// ---- POUs/FB/FB_Licznik.TcPOU
FUNCTION_BLOCK FB_Licznik 
VAR_INPUT
	c_inkrement : BOOL; // sygnal z czujnika
	czas : TIME; // określamy czas, który funkcja czeka po wykryciu butelki,... aby wyeliminowac drgania styków itd. 
END_VAR
VAR_OUTPUT
	c_stan: INT;
END_VAR
VAR
	timer1: TON;
	timer2: TON;
	zbocze	:R_TRIG;
	c_stanpomoc: INT;
END_VAR

c_stanpomoc:=c_stan;

//WHILE c_inkrement:= TRUE DO 					///to może być nie potrzbne 
	timer1(IN := c_inkrement, PT :=T#0.1S);
	zbocze(CLK := timer1.IN);
	IF zbocze.Q THEN
		c_stan:=c_stan+1;
	END_IF		
//END_WHILE

IF c_stan>c_stanpomoc THEN
	timer2(IN := TRUE, PT := czas);
	zbocze(CLK := timer2.IN);
END_IF
c_stanpomoc:=c_stan;

IF GVL_GLOBAL.reset_licznik:= TRUE THEN
	c_stan:=0;
END_IF

END_FUNCTION_BLOCK

// ---- POUs/RecipeManager/RecipeManagement.TcPOU
PROGRAM RecipeManagement
VAR
	fbRecipeManCommands 	: RecipeManCommands; (* Recipe Manager *)
	
	bInit 					: BOOL := TRUE;
	
	nLastError 				: DWORD; (* Error from Recipe Manager *)
	nRecipeCount 			: INT;
	
	sRecipeDef 				: STRING := 'Recipes'; (* current recipe definition *)
	sRecipe 				: STRING; (*Selected recipe *)
	nPreviousIndex			: INT; (* Previous selected index *)
	nPreviousSelectionIndex	: INT := -1; (* *)
	bReload 				: BOOL; (* Refresh recipes from files *)
	fbSaveVariablesTrigger	: R_TRIG;
	bSaveVariables			: BOOL;
	nSelectionIndexInList 	: INT;
	nCount					: INT;
	bReloadValues			: BOOL;
END_VAR

(* Initialization *)
IF bInit THEN
	(* Save the number of recipes in the specified recipe definition in a globar variable.*)
	GVL_RecipeTable.nRecipeCount := fbRecipeManCommands.GetRecipeCount(sRecipeDef);
	
	(* Empty all arrays *)
	FOR nCount := 0 TO cMaxTableRows DO
		GVL_RecipeTable.aRecipeNames[nCount] := '';
		GVL_RecipeTable.aVariableNames[nCount] := '';
		GVL_RecipeTable.aVariableValues[nCount] := '';
	END_FOR
	
	(* save all recipe names of the default recipe definition in an array *)
	fbRecipeManCommands.GetRecipeNames(	sRecipeDef,
										ADR(GVL_RecipeTable.aRecipeNames),
										10,
										GVL_RecipeTable.nRecipeIndex);
										
	GVL_RecipeTable.nRecipeSelectionIndex := -1;
	nPreviousSelectionIndex := -1;
	
	bInit := FALSE;
END_IF

(* Count all recipes in the defined recipe definition *)
nRecipeCount := fbRecipeManCommands.GetRecipeCount(sRecipeDef);
nLastError := fbRecipeManCommands.GetLastError();

(* Scroll position of the recipe list has changed. *)
IF GVL_RecipeTable.nRecipeIndex <> nPreviousIndex THEN
	fbRecipeManCommands.GetRecipeNames(	sRecipeDef,
										ADR(GVL_RecipeTable.aRecipeNames),
										10,
										GVL_RecipeTable.nRecipeIndex);
	nPreviousIndex := GVL_RecipeTable.nRecipeIndex;
END_IF

(* Selection of the current recipe has changed *)
IF GVL_RecipeTable.nRecipeSelectionIndex <> nPreviousSelectionIndex OR bReloadValues THEN
	nPreviousSelectionIndex := GVL_RecipeTable.nRecipeSelectionIndex;
	nSelectionIndexInList := GVL_RecipeTable.nRecipeSelectionIndex - GVL_RecipeTable.nRecipeIndex;
	
	(* Get the selected recipe name *)
	IF nSelectionIndexInList >= 0 AND nSelectionIndexInList < 10 THEN
		sRecipe := GVL_RecipeTable.aRecipeNames[nSelectionIndexInList];
	END_IF
	
	fbRecipeManCommands.GetRecipeValues(sRecipeDef,
										sRecipe,
										ADR(GVL_RecipeTable.aVariableValues),
										10,
										GVL_RecipeTable.nVariableIndex,
										80);
										
	fbRecipeManCommands.GetRecipeVariableNames(	sRecipeDef,
												sRecipe,
												ADR(GVL_RecipeTable.aVariableNames),
												10,
												GVL_RecipeTable.nVariableIndex);
	
	bReloadValues := FALSE;
END_IF

(* Reload the recipe list from the file system *)
IF bReload THEN
	
	fbRecipeManCommands.ReloadRecipes(sRecipeDef);
	bInit := TRUE;
	bReload := FALSE;
END_IF

(* Save the edited values into the recipe *)
fbSaveVariablesTrigger(CLK := bSaveVariables);
IF fbSaveVariablesTrigger.Q THEN
	fbRecipeManCommands.SetRecipeValues(sRecipeDef,
										sRecipe,
										ADR(GVL_RecipeTable.aVariableValues),
										10,
										GVL_RecipeTable.nVariableIndex);	
	bSaveVariables := FALSE;
END_IF

END_PROGRAM

// ---- POUs/Eventy/P_EventsSimple.TcPOU
//==================================================================================================
//							Beckhoff Automation Poland
//									5.2.2016
//		Program sluzy do przesylania globalnych tablic alarmow, ostrzezen i komunikatow do Event Loggera
//  v1.3	|| TC v 3.1.4020.28		|| - poprawki w MESSAGE, dodatkowe komentarze
//  v1.3	|| TC v 3.1.4020.28		|| - kosmetyka
//  v1.2	|| TC v 3.1.4020.28		|| - dodanie MESSAGE
//  v1.1 	|| TC v 3.1.4020.14 	|| - dodanie wersjonowania, komentarzy
// 	v1.0 	|| TC v 3.1.4020.0 		|| - pierwsza wersja
//==================================================================================================
PROGRAM P_EventsSimple
VAR
	fbAlarms				: FB_SimpleEventLog;								// Logowanie alarmow
	fbWarnings				: FB_SimpleEventLog;								// Logowanie ostrzezen
	fbMessage				: FB_SimpleEventLog;								// Logowanie komunikatow
	fbRead1					: FB_AdsReadEvents;									// Odczyt tablicy jezyk polski
	fbRead2					: FB_AdsReadEvents;									// Odczyt tablicy jezyk angielski
	fbRead3					: FB_AdsReadEvents;									// Odczyt tablicy jezyk niemiecki
	fbClear					: ADSCLEAREVENTS;									// Czyszczenie aktywnych alarmow
	MSG_ALARM_ListQuit		: ARRAY[FIRST_MESSAGE..LAST_MESSAGE] OF BOOL;		// Tablica nieuzywana - wymaga potwierdzenia przy usuwaniu
	MSG_MESSAGE_ListQuit	: ARRAY[FIRST_MESSAGE..LAST_MESSAGE] OF BOOL;		// Tablica nieuzywana - wymaga potwierdzenia przy usuwaniu
	MSG_WARNING_ListQuit	: ARRAY[FIRST_MESSAGE..LAST_MESSAGE] OF BOOL;		// Tablica nieuzywana - wymaga potwierdzenia przy usuwaniu
END_VAR

(*
	TCEVENTCLASS_NONE			:=0,	No class
	TCEVENTCLASS_MAINTENANCE	:=1,	Maintenance hint
	TCEVENTCLASS_MESSAGE		:=2,	Message
	TCEVENTCLASS_HINT			:=3,	Hint
	TCEVENTCLASS_STATEINFO		:=4,	State information
	TCEVENTCLASS_INSTRUCTION	:=5,	Instruction
	TCEVENTCLASS_WARNING		:=6,	Warning
	TCEVENTCLASS_ALARM			:=7,	Alarm
	TCEVENTCLASS_PARAMERROR		:=8	 	Parameter error
*)
fbClear(	bClear			:= TRUE,
			iMode			:= TCEVENTLOGIOFFS_CLEARALL);

fbAlarms(	Init			:= TRUE,
			SourceId		:= 1,
			Class			:= TCEVENTCLASS_ALARM,
			QuitRequired	:= FALSE,
			adrAlarmArray	:= ADR(MSG_ALARM_List),
			adrQuitArray	:= ADR(MSG_ALARM_ListQuit));
	
fbWarnings(	Init			:= TRUE,
			SourceId		:= 2,
			Class			:= TCEVENTCLASS_WARNING,
			QuitRequired	:= FALSE,
			adrAlarmArray	:= ADR(MSG_WARNING_List),
			adrQuitArray	:= ADR(MSG_WARNING_ListQuit));

fbMessage(	Init			:= TRUE,
			SourceId		:= 3,
			Class			:= TCEVENTCLASS_MESSAGE,
			QuitRequired	:= FALSE,
			adrAlarmArray	:= ADR(MSG_MESSAGE_List),
			adrQuitArray	:= ADR(MSG_MESSAGE_ListQuit));
			
// Odczyt w kilku jezykach
fbRead1(	bReadEvents		:= TRUE,
			nLanguageId		:= 1045,
			tRefreshTime	:= T#1S);

fbRead2(	bReadEvents		:= TRUE,
			nLanguageId		:= 1033,
			tRefreshTime	:= T#1S);

fbRead3(	bReadEvents		:= TRUE, 
			nLanguageId		:= 1031, 
			tRefreshTime	:= T#1S);
			
// Wybor aktualnego jezyka wyswietlania - przepisanie do tablicy odpowiedniej tablicy
// Uwaga j. polski bez polskich znakow
IF VisuElemsWinControls.CURRENTLANGUAGE		= 'en' THEN
	aEventsSimple			:= fbRead2.aEvents;
ELSIF VisuElemsWinControls.CURRENTLANGUAGE	= 'de' THEN
	aEventsSimple			:= fbRead3.aEvents;
ELSE
	aEventsSimple			:= fbRead1.aEvents;	
END_IF;

END_PROGRAM

// ---- POUs/Eventy/FB_SimpleEventLog.TcPOU
//==================================================================================================
//							Beckhoff Automation Poland
//									22.12.2016
//	Program glowny dla zdarzen wersji advanced
// 	v1.1	|| TC v 3.1.4020.28		|| - idx, ARRAY_LBOUND, ARRAY_UBOUND --> Zmiana typu z UDINT na DINT
// 	v1.0	|| TC v 3.1.4020.28		|| - pierwsza wersja - 13.10.2004, Author:			Dirk Nordberg (BECKHOFF INDUSTRIE ELEKTRONIK)
// Description: Function block to control the EventLogger
// 	Messages can be activated or deactivated through an array of bool.
// 	The subscription of the array is equivalent to EventID from EventLogger.
// 	Funtion block will be initialized with Init flag, then the busy flag is set true. 
// 
// 	Revision:	1.4
// 	History:		13.10.2004	Ng	start coding
// 					17.04.2005	MK	runtime optimized
// 					07.07.2005	MK	short puls BF
// 				    29.11.2010 	MiB  quittierungspflichtige Merker funktionieren nun wieder
///                 21.06.2013  TV   change : data type for pointer address from uint to pointer of int 
//==================================================================================================
///****************************************************************************************
///Name:				FB_SimpleEventLog
///Date:				13.10.2004
// 

FUNCTION_BLOCK FB_SimpleEventLog
VAR_INPUT
	/// Rising flag starts the initialization 
	Init: BOOL;
	/// Number of the source Id 
	SourceId: UINT;
	/// Alarm error class 
	Class: UINT;
	/// Activate or deaktivate confirmation 
	QuitRequired: BOOL;
	/// Adress of the array for the messages 
	adrAlarmArray: POINTER TO BOOL;
	/// ...with constant boundaries ARRAY_LBOUND to ARRAY_UBOUND for array size 
	adrQuitArray: POINTER TO BOOL;
END_VAR
VAR_OUTPUT
	Busy: BOOL;
	Err: BOOL;
	ErrId: UDINT;
END_VAR
VAR CONSTANT
	ARRAY_LBOUND: DINT := FIRST_MESSAGE;
	ARRAY_UBOUND: DINT := LAST_MESSAGE;
	TCEVENTDATAFORMATSTRING: STRING := ' ';
	STATE_INIT: INT := 0;
	STATE_IDLE: INT := 1;
	STATE_RESET_EVENT: INT := 2;
	STATE_QUIT_EVENT: INT := 3;
	STATE_RESET_END: INT := 4;
	STATE_WAIT: INT := 5;
END_VAR
VAR
	state: INT;
	///{flag nowatch on }
	bReady: BOOL := TRUE;
	nMsgHasChanged: DINT;
	bEvtState: ARRAY[ARRAY_LBOUND..ARRAY_UBOUND] OF BOOL;
	event: ARRAY[ARRAY_LBOUND..ARRAY_UBOUND] OF ADSLOGEVENT;
	idx: DINT;
	CfgEvent: TcEvent;
	bWait: BOOL;
	ptAlarm: POINTER TO BOOL;
	ptQuit: POINTER TO BOOL;
	RT_Init: R_TRIG;
END_VAR

nMsgHasChanged := MEMCMP(ADR(bEvtState), adrAlarmArray, SIZEOF(bEvtState));

RT_Init(CLK:=Init);

CASE State OF
	STATE_INIT:		(* Set the parameter for TcEvent *)
		Err := FALSE;
		ErrId :=0;
		Busy := FALSE;
		CfgEvent.Prio := 0;
		CfgEvent.DataFormatStrAddress := ADR(TCEVENTDATAFORMATSTRING);
		// CfgEvent.Flags := TCEVENTFLAG_LOG OR TCEVENTFLAG_SRCID OR TCEVENTFLAG_PRIOCLASS OR TCEVENTFLAG_FMTSELF OR 16#1000;
		// MiB 2015.10.07 Flags changed -> now the class is defined here and not in Event config file.
		CfgEvent.Flags := TCEVENTFLAG_LOG OR TCEVENTFLAG_SRCID;
		CfgEvent.StreamType := TCEVENTSTREAM_SIMPLE;
		CfgEvent.ProgId := 'TcEventFormatter.TcXmlFormatter';
		CfgEvent.SourceId := SourceId;
			CfgEvent.Class := Class ;
		CfgEvent.bQuitRequired := QuitRequired;
		FOR idx := ARRAY_LBOUND TO ARRAY_UBOUND BY 1 DO
			CfgEvent.Id := DINT_TO_UDINT(idx);
			event[idx](NETID:='', PORT:=110, Event:=FALSE , EventQuit:=FALSE,
				 EventConfigData:=CfgEvent, FbCleanup:=FALSE, TMOUT:=t#1s);
		END_FOR;
		State := STATE_IDLE;

	STATE_IDLE:
		(* nothing to do *)
		IF nMsgHasChanged = 0
			AND  NOT QuitRequired
			AND bReady = TRUE
			AND NOT RT_Init.Q THEN
			RETURN;
		END_IF

		IF adrAlarmArray <> 0 THEN
			ptAlarm := adrAlarmArray;
			IF CfgEvent.bQuitRequired AND adrQuitArray <> 0 THEN
				ptQuit := adrQuitArray;
				FOR idx := ARRAY_LBOUND TO ARRAY_UBOUND BY 1 DO
					event[idx](Event:=ptAlarm^, EventQuit:=ptQuit^);
					ptAlarm := ptAlarm + 1;
					ptQuit := ptQuit + 1;
				END_FOR;
				bReady := TRUE;
			ELSE
				bReady := TRUE;
				FOR idx := ARRAY_LBOUND TO ARRAY_UBOUND BY 1 DO
					event[idx](Event:=ptAlarm^);
					IF (NOT (ptAlarm^ = TRUE
							AND event[idx].Event = TRUE		(* event is set/on *)
							AND event[idx].Quit = FALSE
							AND event[idx].EventState = TCEVENTSTATE_SIGNALED)
						AND NOT (ptAlarm^ = FALSE
							AND event[idx].Event = FALSE		(* event is reset/off *)
							AND event[idx].Quit = TRUE
							AND event[idx].EventState = TCEVENTSTATE_INVALID)) THEN
						bReady := FALSE;
					END_IF
					ptAlarm := ptAlarm + 1;
				END_FOR;

				(* copy the status *)
				IF bReady THEN
					MEMCPY(ADR(bEvtState), adrAlarmArray, SIZEOF(bEvtState));
				END_IF

			END_IF
		END_IF

		IF RT_Init.Q THEN
			Busy := TRUE;
			State := STATE_RESET_EVENT;
		END_IF

	STATE_RESET_EVENT:(*---------------------------------- clear messages ----------------------------------------*)
		FOR idx := ARRAY_LBOUND TO ARRAY_UBOUND BY 1 DO
			IF event[idx].EventState = TCEVENTSTATE_SIGNALED THEN
				event[idx](Event:=FALSE, EventQuit:= FALSE, FbCleanup:= FALSE, TMOUT:= t#1s);
				IF event[idx].Err THEN
					Err := TRUE;
					ErrId := event[idx].ErrId;
					IF event[idx].ErrId = 1282 THEN	(* Message Router: mailbox full *)
						event[idx](Event:=FALSE, EventQuit:= FALSE, FbCleanup:= FALSE);
						RETURN;
					END_IF
				END_IF
			END_IF;
		END_FOR;
		State := STATE_QUIT_EVENT;

	STATE_QUIT_EVENT:(*---------------------------------- quit messages ----------------------------------------*)
		FOR idx := ARRAY_LBOUND TO ARRAY_UBOUND BY 1 DO
			IF event[idx].EventState = TCEVENTSTATE_SIGNALED THEN
				event[idx](Event:=FALSE, EventQuit:= TRUE, FbCleanup:= FALSE, TMOUT:= t#1s);
				IF event[idx].Err THEN
					Err := TRUE;
					ErrId := event[idx].ErrId;
					IF event[idx].ErrId = 1282 THEN	(* Message Router: mailbox full *)
						event[idx](Event:=FALSE, EventQuit:= FALSE, FbCleanup:= FALSE);
						RETURN;
					END_IF
				END_IF
			END_IF;
		END_FOR;
		State := STATE_RESET_END;

	STATE_RESET_END:
		bWait := FALSE;
		FOR idx := ARRAY_LBOUND TO ARRAY_UBOUND BY 1 DO
			event[idx](Event:=FALSE, EventQuit:= FALSE, FbCleanup:= FALSE);
			IF event[idx].EventState = TCEVENTSTATE_SIGNALED THEN
				bWait := TRUE;
			END_IF
		END_FOR;
		IF NOT bWait THEN
			State := STATE_INIT;
		END_IF

END_CASE

END_FUNCTION_BLOCK

// ---- POUs/FB/FB_INV000_MX2_Alarm.TcPOU
FUNCTION_BLOCK FB_INV000_MX2_Alarm
VAR_INPUT
	Enable							:BOOL;	
	Fault_Monitor_1_Inverter_Status	:UINT;
	Fault_Monitor_1_Cause			:UINT;	
	Status							:WORD;	

END_VAR
VAR_OUTPUT
	ENO								:BOOL;	
	Alarm_Status					:STRING[256];
	Alarm_Fault						:STRING[256];	

END_VAR
VAR
	tmp_Status						:uWORD_BOOL_MX2;
END_VAR

///FB ON///
ENO:=Enable;

///Status extraction///
	tmp_Status.ch := Status;

//If MX2 has an fault the latest fault will be outputted//
IF tmp_Status.bits[3]=TRUE THEN
	
//MX2 Inverter fault factor list name//
CASE Fault_Monitor_1_Cause OF
	00 : 
		Alarm_Fault:='No trip factor';	
	01 : 
		Alarm_Fault:='Overcurrent protection during constant speed';
   	02 : 
		Alarm_Fault:='Overcurrent protection during deceleration';
	03 : 
		Alarm_Fault:='Overcurrent protection during acceleration';
	04 : 
		Alarm_Fault:='Overcurrent protection during stop';
	05 : 
		Alarm_Fault:='Overload protection';
	06 : 
		Alarm_Fault:='Braking resistor overload protection';
	07 : 
		Alarm_Fault:='Overvoltage protection';
	08 : 
		Alarm_Fault:='EEPROM error';
	09 : 
		Alarm_Fault:='Undervoltage protection';
	10 : 
		Alarm_Fault:='Current detector error';
	11 : 
		Alarm_Fault:='CPU error';
	12 : 
		Alarm_Fault:='External trip';
	13 : 
		Alarm_Fault:='USP error';
	14 : 
		Alarm_Fault:='Grounding protection';
	15 : 
		Alarm_Fault:='Incoming overvoltage protection';
	21 : 
		Alarm_Fault:='Abnormal temperature';
	25 : 
		Alarm_Fault:='Main circuit error';
	30 : 
		Alarm_Fault:='Driver error';
	35 : 
		Alarm_Fault:='Thermistor error';
	36 : 
		Alarm_Fault:='Brake error';
	37 : 
		Alarm_Fault:='Emergency shutoff';
	38 : 
		Alarm_Fault:='Overload protection in a low speed range';
	40 : 
		Alarm_Fault:='Digital operator connection error';
	41 : 
		Alarm_Fault:='Modbus communication (Modbus-RTU) error';
	43..45 : 
		Alarm_Fault:='Internal data error';
	50..69 : 
		Alarm_Fault:='Internal data error';	
	80 : 
		Alarm_Fault:='Encoder disconnection';
	81 : 
		Alarm_Fault:='Overspeed';
	83 : 
		Alarm_Fault:='Position control range trip';
	

		
END_CASE;

//MX2 Inverter status at fault occur//


	CASE Fault_Monitor_1_Inverter_Status OF
    	0 : 
			Alarm_Status:='During reset';
		1 : 
			Alarm_Status:='During stop';
		2 : 
			Alarm_Status:='During deceleration';
		3 : 
			Alarm_Status:='At a constant speed';
		4 : 
			Alarm_Status:='During acceleration';
		5 : 
			Alarm_Status:='Operates at frequency = 0';
		6 : 
			Alarm_Status:='During startup';
		7 : 
			Alarm_Status:='DB active (DC injection braking active)';
		8 : 
			Alarm_Status:='During overload limit';
		
	END_CASE;
ELSE
	Alarm_Fault:='No trip factor';	
	Alarm_Status:='--';
	
END_IF;

END_FUNCTION_BLOCK

// ---- POUs/FB/FB_INV003_MX2_ECT.TcPOU
FUNCTION_BLOCK FB_INV003_MX2_ECT
VAR_INPUT
	Output_Frequency_Monitor						:UINT;
	Enable											:BOOL;
	Fwd												:BOOL;	
	Rev												:BOOL;	
	Fault_Reset										:BOOL;	
	Frequency_in									:REAL;	
	Acceleration									:REAL;		
	Deceleration									:REAL;	
END_VAR
VAR_OUTPUT
	ENO												:BOOL;
	Frequency_out									:REAL;	
	During_Fwd										:BOOL;
	During_Rev										:BOOL;	
	Fault											:BOOL;		
	Warning											:BOOL;		
	Remote											:BOOL;	
	Freq_Match										:BOOL;	
	Connection_Error								:BOOL;		
END_VAR
VAR
	tmp_freq_in_real								:REAL;
	tmp_freq_in_int									:UINT;			
	tmp_freq_out_real								:REAL;			
	tmp_freq_out_int								:UINT;			
	tmp_acc_real									:REAL;				
	tmp_acc_int										:INT;				
	tmp_dec_real									:REAL;				
	tmp_dec_int										:INT;		
	tmp_Command										:uWORD_BOOL_MX2;			
	tmp_Status										:uWORD_BOOL_MX2;	
END_VAR
VAR_IN_OUT
	Command												:WORD;	
	Frequency_Reference									:UINT;	
	F002_1st_Acceleration								:UDINT;		
	F003_1st_Deceleration								:UDINT;		
	Status												:WORD;	
END_VAR

///Status extraction///
	tmp_Status.ch := Status;
	During_Fwd := tmp_Status.bits[0];
	During_Rev := tmp_Status.bits[1];
	Fault := tmp_Status.bits[3];
	Warning := tmp_Status.bits[7];
	Remote := tmp_Status.bits[9];
	Freq_Match := tmp_Status.bits[12];
	Connection_Error := tmp_Status.bits[15];

///Command extraction///
IF Enable THEN;
	tmp_Command.bits[0] := Fwd;
	tmp_Command.bits[1] := Rev;
	ENO:=TRUE;
ELSE
	tmp_Command.bits[0] := FALSE;
	tmp_Command.bits[1] := FALSE;
	ENO:=FALSE;
END_IF;
	tmp_Command.bits[7] := Fault_Reset;
	Command := tmp_Command.ch;

///Frequence form a REAL value///
IF Frequency_in>0.01 THEN;
	tmp_freq_in_real:=Frequency_in*100;
	tmp_freq_in_int:=REAL_TO_UINT(tmp_freq_in_real);
	Frequency_Reference:=tmp_freq_in_int;
END_IF;

//Convert Output_Frequency_Monitor to a REAL value//
	tmp_freq_out_int:=Output_Frequency_Monitor;
	tmp_freq_out_real:=UINT_TO_REAL(tmp_freq_out_int);
	Frequency_out:=tmp_freq_out_real/100.0;
	
//Acceleration/Deceleration Time  in REAL value//
IF Acceleration>0.01 THEN;
	tmp_acc_real:=Acceleration*100;
	tmp_acc_int:=REAL_TO_INT(tmp_acc_real);
	F002_1st_Acceleration:=tmp_acc_int;
END_IF;

IF Deceleration>0.01 THEN;
	tmp_dec_real:=Deceleration*100;
	tmp_dec_int:=REAL_TO_INT(tmp_dec_real);
	F003_1st_Deceleration:=tmp_dec_int;
END_IF;

END_FUNCTION_BLOCK

// ---- POUs/Programy/Hbot/AxisOnline/POUsAxisOnline/AX5000/FB_AxisDiag_1.TcPOU
//==================================================================================================
//							Beckhoff Automation Poland
//								23.05.2018
//					Blok do diagnostyki osi
// 	v1.1	|| TC v 3.1.4022.16	|| - optymalizacja kodu
// 	v1.0	|| TC v 3.1.4020.0	|| - pierwsza wersja
//==================================================================================================
FUNCTION_BLOCK FB_AxisDiag_1
VAR_INPUT
	IPCNetID							: T_AmsNetId; 	(* AmsNetId of the IPC *)
	Timeout								: TIME := DEFAULT_ADS_TIMEOUT;
	Reset								: BOOL;
	GetDiag								: BOOL;
END_VAR
VAR_IN_OUT
	Axis	 							: AXIS_REF;
	stAX5000Diag						: ST_AX5000Diag;
END_VAR
VAR_OUTPUT
	Error								: BOOL;
	AdsErrId							: UINT;
	SercosErrId							: UINT;
	ResetAct							: BOOL;
	DiagAct								: BOOL;
	Busy								: BOOL;
END_VAR
VAR
	iState								: INT;
	iSubState							: INT;
	GetDriveRef							: BOOL;
	DriveRef								: ST_DriveRef; (* contains sNetID of EcMaster, nSlaveAddr of EcDrive, nDriveNo of EcDrive, either preset or read from NC *)
	AxisID								: UDINT;

	C1DErrorPrev							: BOOL;
	WcStateErrorPrev						: BOOL;
	AxisErrorPrev							: BOOL;
	OperationalPrev						: BOOL;
	ResetPrev							: BOOL;
	GetDiagPrev							: BOOL;

	fbSoERead							: FB_SoERead;
	fbDiagMessage 						: FB_SoEReadDiagMessage;
	fbClassXDiag							: FB_SoEReadClassXDiag;
	fbDiagNumber						: FB_SoEReadDiagNumber;
	fbDiagNumberList						: FB_SoEReadDiagNumberList;

	fbReset								: FB_SoEReset;
	fbDelay								: TON;
	fbGetSlaveState 						: FB_EcGetSlaveState;
	fbReqSlaveState 						: FB_EcReqSlaveState;
	fbNcReset 							: MC_Reset;

	fbAdsRead							: ADSREAD;
	readBuffer							: ARRAY[0..9] OF BYTE;
	Ids									: T_AmsNetIdArr;
	strSoEString							: ST_SoE_String;
END_VAR
VAR CONSTANT
	NCIDXG_AXPARMS					: UDINT := 16#00004000;	(* Axis with ID: Parameter 			*)
	NCIDXO_AXP_HWAMSADDR			: UDINT := 16#00000031;
END_VAR

stAX5000Diag.bOperational	:= Axis.NcToPlc.StateDWord.0;
stAX5000Diag.bC1DError	 	:= Axis.NcToPlc.StateDWord.28;
stAX5000Diag.bWcStateError 	:= Axis.NcToPlc.StateDWord.30;
stAX5000Diag.bAxisError		:= Axis.NcToPlc.StateDWord.31;
stAX5000Diag.iAxisErrorCode	:= Axis.NcToPlc.ErrorCode;

CASE iState OF
0:	(* idle *)
	GetDriveRef 	:= (DriveRef.nSlaveAddr = 0);

	IF GetDriveRef THEN
		Busy			:= TRUE;
		Error			:= FALSE;
		AdsErrId		:= 0;
		SercosErrId		:= 0;
		iState 			:= 1;
		iSubState		:= 0;
		AxisID 			:= Axis.NcToPlc.AxisId;

	ELSIF Reset AND NOT ResetPrev THEN
		Busy			:= TRUE;
		ResetAct		:= TRUE;
		ResetPrev		:= Reset;
		Error			:= FALSE;
		AdsErrId		:= 0;
		SercosErrId		:= 0;
		iState 			:= 2;
		iSubState		:= 0;
		AxisID 			:= Axis.NcToPlc.AxisId;

	ELSIF GetDiag AND NOT GetDiagPrev OR
		(stAX5000Diag.bC1DError AND NOT C1DErrorPrev) OR (NOT stAX5000Diag.bC1DError AND C1DErrorPrev) (* rising/falling C1D *) OR
		(stAX5000Diag.bWcStateError AND NOT WcStateErrorPrev) OR (NOT stAX5000Diag.bWcStateError AND WcStateErrorPrev) (* rising/falling WcState *) OR
		(stAX5000Diag.bAxisError AND NOT AxisErrorPrev) OR (NOT stAX5000Diag.bAxisError AND AxisErrorPrev) (* rising/falling NcError *) OR
		(stAX5000Diag.bOperational AND NOT OperationalPrev) OR (NOT stAX5000Diag.bOperational AND OperationalPrev) (* rising/falling Enable *) THEN

		Busy			:= TRUE;
		DiagAct			:= TRUE;
		GetDiagPrev		:= GetDiag;
		Error			:= FALSE;
		AdsErrId		:= 0;
		SercosErrId		:= 0;
		iState 			:= 3;
		iSubState		:= 0;
		AxisID 			:= Axis.NcToPlc.AxisId;

		(* set/clear flags *)
		C1DErrorPrev		:= stAX5000Diag.bC1DError;
		WcStateErrorPrev	:= stAX5000Diag.bWcStateError;
		AxisErrorPrev		:= stAX5000Diag.bAxisError;
		OperationalPrev		:= stAX5000Diag.bOperational;

	ELSE
		ResetAct	:= FALSE;
		DiagAct		:= FALSE;
	END_IF

1:	(* get drive reference *)
	M_GetDriveRef();

2:	(* reset and state change *)
	M_Reset();

3:	(* get diag data *)
	M_GetDiagnosis();

END_CASE

(* clear latch *)
ResetPrev	:= ResetPrev AND Reset;
GetDiagPrev	:= GetDiagPrev AND GetDiag;

ACTION M_GetDiagnosis:
CASE iSubState OF
0:	fbClassXDiag(
		NetId		:= IPCNetID,
		Execute		:= TRUE,
		DiagClass 	:= 1,
		Timeout		:= DEFAULT_ADS_TIMEOUT,
		Axis		:= Axis,
	);

	IF NOT fbClassXDiag.Busy THEN
		fbClassXDiag(Execute:= FALSE,Axis := Axis);

		IF NOT fbClassXDiag.Error THEN
			stAX5000Diag.wClass1Diag	:= fbClassXDiag.ClassXDiag;
			stAX5000Diag.stClass1Diag	:= F_ConvWordToSTAX5000C1D(stAX5000Diag.wClass1Diag);
		ELSE
			Error			:= TRUE;
			AdsErrId		:= fbClassXDiag.AdsErrId;
			SercosErrId	:= fbClassXDiag.SercosErrId;
		END_IF
		iSubState	:= iSubState + 1;
	END_IF

1:	fbDiagMessage(
		NetId	:= IPCNetID,
		Execute	:= TRUE,
		Timeout	:= DEFAULT_ADS_TIMEOUT,
		Axis	:= Axis,
	);

	IF NOT fbDiagMessage.Busy THEN
		fbDiagMessage(Execute:= FALSE,Axis := Axis);

		IF NOT fbDiagMessage.Error THEN
			stAX5000Diag.strDiagMessage := LEFT(fbDiagMessage.DiagMessage.strData, UINT_TO_INT(fbDiagMessage.DiagMessage.iActualSize));
		ELSE
			Error			:= TRUE;
			AdsErrId		:= fbDiagMessage.AdsErrId;
			SercosErrId	:= fbDiagMessage.SercosErrId;
		END_IF
		iSubState	:= iSubState + 1;
	END_IF

2:	fbDiagNumber(
		NetId	:= IPCNetID,
		Execute	:= TRUE,
		Timeout	:= DEFAULT_ADS_TIMEOUT,
		Axis	:= Axis,
	);

	IF NOT fbDiagNumber.Busy THEN
		fbDiagNumber(Execute:= FALSE,Axis := Axis);

		IF NOT fbDiagNumber.Error THEN
			stAX5000Diag.iDiagNumber := fbDiagNumber.DiagNumber;
		ELSE
			Error			:= TRUE;
			AdsErrId		:= fbDiagNumber.AdsErrId;
			SercosErrId	:= fbDiagNumber.SercosErrId;
		END_IF
		iSubState	:= iSubState + 1;
	END_IF

3:	fbSoERead(
		NetId	:= IPCNetID,
		Execute	:= TRUE,
		Idn		:= 135,
		Element	:=16#44,
		pDstBuf	:=ADR(stAX5000Diag.wDriveStatus),
		BufLen	:=SIZEOF(stAX5000Diag.wDriveStatus),
		Timeout	:= DEFAULT_ADS_TIMEOUT,
		Axis	:= Axis,
	);

	IF NOT fbSoERead.Busy THEN
		fbSoERead(Execute:= FALSE,Axis := Axis);
		IF NOT fbSoERead.Error THEN
			stAX5000Diag.stDriveStatus := F_ConvWordToSTAX5000DriveStatus(stAX5000Diag.wDriveStatus);
			iSubState		:= iSubState + 1;
		ELSE
			Error			:= TRUE;
			AdsErrId		:= fbSoERead.AdsErrId;
			SercosErrId	:= fbSoERead.SercosErrId;
			iSubState		:= iSubState + 2;
		END_IF
	END_IF

4:	fbSoERead(
		NetId	:= IPCNetID,
		Execute	:= TRUE,
		Idn		:= stAX5000Diag.stDriveStatus.iActOpModeParNum,
		Element	:=16#44,
		pDstBuf	:=ADR(stAX5000Diag.stDriveStatus.eActOpMode),
		BufLen	:=SIZEOF(stAX5000Diag.stDriveStatus.eActOpMode),
		Timeout	:= DEFAULT_ADS_TIMEOUT,
		Axis	:= Axis,
	);

	IF NOT fbSoERead.Busy THEN
		fbSoERead(Execute:= FALSE,Axis := Axis);
		IF NOT fbSoERead.Error THEN
			;
		ELSE
			Error			:= TRUE;
			AdsErrId		:= fbSoERead.AdsErrId;
			SercosErrId	:= fbSoERead.SercosErrId;
		END_IF
		iSubState	:= iSubState + 1;
	END_IF

5:	fbGetSlaveState(
		sNetId		:= DriveRef.sNetId,
		nSlaveAddr	:= DriveRef.nSlaveAddr,
		bExecute	:= TRUE,
		tTimeout	:= DEFAULT_ADS_TIMEOUT,
	);

	IF NOT fbGetSlaveState.bBusy THEN
		fbGetSlaveState(bExecute:= FALSE);
		IF NOT fbGetSlaveState.bError THEN
			stAX5000Diag.stEcSlaveState := fbGetSlaveState.state;
			stAX5000Diag.stEcSlaveStateBits := F_ConvSlaveStateToBits(fbGetSlaveState.state);
		ELSE
			Error			:= TRUE;
			AdsErrId		:= UDINT_TO_UINT(fbGetSlaveState.nErrId);
		END_IF

		IF stAX5000Diag.stEcSlaveStateBits.bError THEN
			IF stAX5000Diag.stEcSlaveStateBits.bPreop THEN
				(* read S21 - IDN List of Invalid operation data for CP2 (Preop->SaveOp) *)
				MEMSET(ADR(stAX5000Diag.stCPxInvParamList), 0, SIZEOF(stAX5000Diag.stCPxInvParamList));
				stAX5000Diag.bPreopToSafeOpError := TRUE;
				stAX5000Diag.bSafeOpToOpError := FALSE;
				iSubState	:= iSubState + 1;
			ELSIF stAX5000Diag.stEcSlaveStateBits.bSafeOp THEN
				(* read S22 - IDN List of Invalid operation data for CP3 (SaveOp->Op) *)
				MEMSET(ADR(stAX5000Diag.stCPxInvParamList), 0, SIZEOF(stAX5000Diag.stCPxInvParamList));
				stAX5000Diag.bPreopToSafeOpError := FALSE;
				stAX5000Diag.bSafeOpToOpError := TRUE;
				iSubState	:= iSubState + 2;
			ELSE
				(* Skip S21 + S22 *)
				MEMSET(ADR(stAX5000Diag.stCPxInvParamList), 0, SIZEOF(stAX5000Diag.stCPxInvParamList));
				stAX5000Diag.bPreopToSafeOpError := FALSE;
				stAX5000Diag.bSafeOpToOpError := FALSE;
				iSubState	:= iSubState + 3;
			END_IF
		ELSE
			(* Skip S21 + S22 *)
			MEMSET(ADR(stAX5000Diag.stCPxInvParamList), 0, SIZEOF(stAX5000Diag.stCPxInvParamList));
			stAX5000Diag.bPreopToSafeOpError := FALSE;
			stAX5000Diag.bSafeOpToOpError := FALSE;
			iSubState	:= iSubState + 3;
		END_IF
	END_IF

6:	(* read S21 - IDN List of Invalid operation data for CP2 (Preop->SaveOp) *)
	fbSoERead(
		NetId	:= IPCNetID,
		Execute	:= TRUE,
		Idn		:= 21,
		Element	:=16#40,
		pDstBuf	:=ADR(stAX5000Diag.stCPxInvParamList),
		BufLen	:=SIZEOF(stAX5000Diag.stCPxInvParamList),
		Timeout	:= DEFAULT_ADS_TIMEOUT,
		Axis	:= Axis,
	);

	IF NOT fbSoERead.Busy THEN
		fbSoERead(Execute:= FALSE,Axis := Axis);
		IF NOT fbSoERead.Error THEN
			;
		ELSE
			Error			:= TRUE;
			AdsErrId		:= fbSoERead.AdsErrId;
			SercosErrId	:= fbSoERead.SercosErrId;
		END_IF
		iSubState	:= iSubState + 2;
	END_IF

7:	(* read S22 - IDN List of Invalid operation data for CP3 (SaveOp->Op) *)
	fbSoERead(
		NetId	:= IPCNetID,
		Execute	:= TRUE,
		Idn		:= 22,
		Element	:=16#40,
		pDstBuf	:=ADR(stAX5000Diag.stCPxInvParamList),
		BufLen	:=SIZEOF(stAX5000Diag.stCPxInvParamList),
		Timeout	:= DEFAULT_ADS_TIMEOUT,
		Axis	:= Axis,
	);

	IF NOT fbSoERead.Busy THEN
		fbSoERead(Execute:= FALSE,Axis := Axis);
		IF NOT fbSoERead.Error THEN
			;
		ELSE
			Error			:= TRUE;
			AdsErrId		:= fbSoERead.AdsErrId;
			SercosErrId	:= fbSoERead.SercosErrId;
		END_IF
		iSubState	:= iSubState + 1;
	END_IF

8:	fbDiagNumberList(
		NetId			:= IPCNetID,
		Execute			:= TRUE,
		Timeout			:= DEFAULT_ADS_TIMEOUT,
		pDiagNumber		:= ADR(stAX5000Diag.stDiagNumberList),
		Size			:= SIZEOF(stAX5000Diag.stDiagNumberList),
		Axis			:= Axis,
	);

	IF NOT fbDiagNumberList.Busy THEN
		fbDiagNumberList(Execute:= FALSE,Axis := Axis);

		IF fbDiagNumberList.Error THEN
			Error			:= TRUE;
			AdsErrId		:= fbDiagNumberList.AdsErrId;
			SercosErrId	:= fbDiagNumberList.SercosErrId;
		END_IF

		IF (stAX5000Diag.strMotorType = '') OR (stAX5000Diag.strDriveType = '') THEN
			iSubState	:= iSubState + 1;
		ELSE
			DiagAct	:= FALSE;
			iSubState	:= 0;
			iState		:= 0;
			Busy		:= FALSE;
		END_IF
	END_IF

9:	fbSoERead(
		NetId	:= IPCNetID,
		Execute	:= TRUE,
		Idn		:= P_0_IDN + 53,
		Element	:=16#44,
		pDstBuf	:=ADR(strSoEString),
		BufLen	:=SIZEOF(strSoEString),
		Timeout	:= DEFAULT_ADS_TIMEOUT,
		Axis	:= Axis,
	);

	IF NOT fbSoERead.Busy THEN
		fbSoERead(Execute:= FALSE,Axis := Axis);
		IF NOT fbSoERead.Error THEN
			MEMSET(ADR(stAX5000Diag.strMotorType),0,SIZEOF(stAX5000Diag.strMotorType));
			MEMCPY(ADR(stAX5000Diag.strMotorType),ADR(strSoEString.strData),MIN(SIZEOF(stAX5000Diag.strMotorType),strSoEString.iActualSize));
		ELSE
			Error			:= TRUE;
			AdsErrId		:= fbSoERead.AdsErrId;
			SercosErrId	:= fbSoERead.SercosErrId;
		END_IF
		iSubState	:= iSubState + 1;
	END_IF

10:	fbSoERead(
		NetId	:= IPCNetID,
		Execute	:= TRUE,
		Idn		:= P_0_IDN + 324,
		Element	:=16#44,
		pDstBuf	:=ADR(strSoEString),
		BufLen	:=SIZEOF(strSoEString),
		Timeout	:= DEFAULT_ADS_TIMEOUT,
		Axis	:= Axis,
	);

	IF NOT fbSoERead.Busy THEN
		fbSoERead(Execute:= FALSE,Axis := Axis);
		IF NOT fbSoERead.Error THEN
			MEMSET(ADR(stAX5000Diag.strDriveType),0,SIZEOF(stAX5000Diag.strDriveType));
			MEMCPY(ADR(stAX5000Diag.strDriveType),ADR(strSoEString.strData),MIN(SIZEOF(stAX5000Diag.strDriveType),strSoEString.iActualSize));
		ELSE
			Error			:= TRUE;
			AdsErrId		:= fbSoERead.AdsErrId;
			SercosErrId	:= fbSoERead.SercosErrId;
		END_IF
		DiagAct	:= FALSE;
		iSubState	:= 0;
		iState		:= 0;
		Busy		:= FALSE;
	END_IF


END_CASE
END_ACTION

ACTION M_GetDriveRef:
(* get reference from NC *)
fbAdsRead(
	NETID	:= IPCNetID,
	PORT	:= AMSPORT_R0_NC,
	IDXGRP	:= NCIDXG_AXPARMS + Axis.NcToPlc.AxisId,
	IDXOFFS	:= NCIDXO_AXP_HWAMSADDR,
	LEN		:= SIZEOF(readBuffer) ,
	DESTADDR:= ADR(readBuffer),
	READ	:= TRUE,
	TMOUT	:= Timeout
);

IF NOT fbAdsRead.BUSY THEN
	fbAdsRead(READ := FALSE);
	stAX5000Diag.nNCAxisID := Axis.NcToPlc.AxisId;

	IF NOT fbAdsRead.ERR THEN
		MEMCPY(ADR(Ids), ADR(readBuffer), SIZEOF(Ids)); 										(* readBuffer[0..5] *)
		MEMCPY(ADR(DriveRef.nSlaveAddr), ADR(readBuffer[6]), SIZEOF(DriveRef.nSlaveAddr));  	(* readBuffer[6..7] *)
		MEMCPY(ADR(DriveRef.nDriveNo), ADR(readBuffer[8]), SIZEOF(DriveRef.nDriveNo));  		(* readBuffer[8..9] *)

		(* create string out of byte array *)
		DriveRef.sNetId := F_CreateAmsNetId(Ids);
		GetDriveRef := FALSE;
	END_IF

	Busy	:= FALSE;
	iState	:= 0;
END_IF
END_ACTION

ACTION M_Reset:
CASE iSubState OF
0:
	IF stAX5000Diag.bWcStateError OR stAX5000Diag.bC1DError THEN
		(* ResetAmplifier *)
		iSubState := iSubState + 1;
	ELSIF (NOT stAX5000Diag.bOperational) OR stAX5000Diag.bAxisError OR (stAX5000Diag.iAxisErrorCode <> 0) THEN
		(* NC Reset only *)
		iSubState := 6;
	ELSE
		(* reset not required *)
		iSubState	:= 0;
		iState		:= 0;
		Busy		:= FALSE;
		ResetAct	:= FALSE;
	END_IF

1:	(* ResetAmplifier *)
	fbReset(
		NetId	:= IPCNetID,
		Execute	:= TRUE,
		Timeout	:= DEFAULT_ADS_TIMEOUT,
		Axis	:= Axis,
	);
	IF NOT fbReset.Busy THEN
		fbReset(Execute:= FALSE, Axis:= Axis);

		IF NOT fbReset.Error THEN
			iSubState	:= iSubState + 1;
		ELSE
			Error			:= TRUE;
			AdsErrId		:= fbReset.AdsErrId;
			SercosErrId		:= fbReset.SercosErrId;
			Busy			:= FALSE;
			ResetAct		:= FALSE;
			iSubState		:= 0;
			iState			:= 0;
		END_IF
	END_IF

2:	fbDelay(IN:=TRUE, PT:=t#3s);
	IF fbDelay.Q THEN
		fbDelay(IN:=FALSE);
		iSubState	:= iSubState + 1;
	END_IF

3:	fbGetSlaveState(
		sNetId		:= DriveRef.sNetId,
		nSlaveAddr	:= DriveRef.nSlaveAddr,
		bExecute	:= TRUE,
		tTimeout	:= DEFAULT_ADS_TIMEOUT,
	);

	IF NOT fbGetSlaveState.bBusy THEN
		fbGetSlaveState(bExecute:= FALSE);

		IF NOT fbGetSlaveState.bError THEN
			IF Axis.NcToPlc.StateDWord.31 OR (Axis.NcToPlc.ErrorCode <> 0) THEN
				iSubState	:= 6;
			ELSE
				Busy		:= FALSE;
				ResetAct	:= FALSE;
				iSubState	:= 0;
				iState		:= 0;
			END_IF
		ELSE
			Error			:= TRUE;
			AdsErrId		:= UDINT_TO_UINT(fbGetSlaveState.nErrId);
			Busy			:= FALSE;
			ResetAct		:= FALSE;
			iSubState		:= 0;
			iState			:= 0;
		END_IF
	END_IF

5:	(* set op *)
	fbReqSlaveState(
		sNetId		:= DriveRef.sNetId,
		nSlaveAddr	:= DriveRef.nSlaveAddr,
		bExecute	:= TRUE,
		tTimeout	:= DEFAULT_ADS_TIMEOUT,
		state		:= EC_DEVICE_STATE_OP);

	IF NOT fbReqSlaveState.bBusy THEN
		fbReqSlaveState(bExecute:= FALSE);

		IF NOT fbReqSlaveState.bError THEN
			iSubState	:= iSubState + 1;
		ELSE
			Error		:= TRUE;
			AdsErrId	:= UDINT_TO_UINT(fbReqSlaveState.nErrId);
			Busy		:= FALSE;
			ResetAct	:= FALSE;
			iSubState	:= 0;
			iState		:= 0;
		END_IF
	END_IF

6:	fbNcReset(
		Execute:= TRUE,
		Axis:= Axis,
	);
	IF fbNcReset.Done OR fbNcReset.Error THEN
		IF fbNcReset.Error THEN
			Error 		:= TRUE;
			AdsErrId 	:= UDINT_TO_UINT(fbNcReset.ErrorID);
		END_IF

		iSubState	:= 0;
		iState		:= 0;
		Busy		:= FALSE;
		ResetAct	:= FALSE;
		fbNcReset(Execute:= FALSE, Axis:= Axis);
	END_IF
END_CASE
END_ACTION

END_FUNCTION_BLOCK

// ---- POUs/Programy/Hbot/NCI/2_GROUPS/FB_ReleaseAllGroups.TcPOU
FUNCTION_BLOCK FB_ReleaseAllGroups
VAR_INPUT
	bExec: 				BOOL;
END_VAR
VAR_OUTPUT
	bBusy: 				BOOL;
	bErr: 				BOOL;
	nErrId:				UDINT:=0;
END_VAR
VAR
	nState: 				UINT;
	i: 					UINT;
	fbReleaseGroup:	FB_ReleaseGroup;
	nChan: 				UINT;
	bInterIdle: 		BOOL;
	nItpState: 			UDINT;
	fbRtrig: 			R_TRIG;
END_VAR

(* ==========================================================*)
(*   FB: FB_ReleaseAllGroups	                             *)
(* ----------------------------------------------------------*)
(*   Desc: Release all axis from all groups                  *)
(*   Auth: MiB  / TV                                         *)
(*   Date: 02.09.2005                                        *)
(*   Last: 02.04.2013                                        *)
(*   Rev.: 1.1                                               *)
(* ==========================================================*)

fbRtrig(Clk := bExec);

CASE nState OF
16#0: (* init *)
		IF fbRtrig.Q THEN
			bBusy	:= TRUE;
			bErr	:= FALSE;
			nErrId	:= 0;
			nState := 16#10;
			nChan := 2;       (* first NCI channel is channel 2 *)
			bInterIdle := TRUE;
		END_IF

16#10: (* check if channels in IDLE state *)
		FOR  i:=1 TO nMaxNumberOfNciChannels DO
			nItpState := arrNCToPLC_NCIChannel_REF[i].ItpState;
			IF (nItpState <> NCI_INTERPRETER_IDLE) THEN
				bInterIdle := FALSE;
			END_IF
		END_FOR
		IF NOT bInterIdle THEN  (* cannot start releasing groups, while interpreter is not in IDLE mode *)
			nState := 16#999;
			nErrId := 16#10;
		ELSE
			nState := 16#20;   (* release groups *)
		END_IF


16#20: (* Realease all groups in all Channels > 1*)
		fbReleaseGroup(
					bExec:=TRUE ,
					nChan:=nChan,
					bBusy=> ,
					bErr=> ,
					nErrId=> );
		IF NOT fbReleaseGroup.bBusy THEN
			fbReleaseGroup( bExec := FALSE );
			nChan := nChan + 1;
			IF (fbReleaseGroup.bErr) THEN
				(* an error occured *)
				nErrId	:= fbReleaseGroup.nErrId;
				nState	:= 16#999;
			ELSE
				IF (nChan-1) > nMaxNumberOfNciChannels THEN
					nState := 16#30;
				END_IF
			END_IF
		END_IF


16#30:	(* Ready *)

	bBusy := FALSE;
	nState := 0;

16#999:  (* Error *)
	bBusy := FALSE;
	bErr		:= TRUE;
	nState := 0;
		;
END_CASE

END_FUNCTION_BLOCK

// ---- POUs/Programy/PRG_CaseErector.TcPOU
PROGRAM PRG_CaseErector

(*----------------------------------------------NOWE Wejściowe ------------------------------------------*)
VAR_INPUT
	eMachineMode							: E_LineMachineMode; 		// Machine mode
	eMachineCommand							: E_LineMachineCommand; 	// Command from top level state program
END_VAR
(*----------------------------------------------NOWE Wyjściowe ------------------------------------------*)
VAR_OUTPUT
	eMachineState							: E_CaseErectorMachineState;
  	bError									: BOOL;
END_VAR
(*----------------------------------------------NOWE Wewnętrzne ------------------------------------------*)
VAR
	// INPUTS
	bIn1									: BOOL;
	// OUTPUTS
	bOut1									: BOOL;	
	// Local
	iStateIdle								: INT;
	iStepStarting							: INT;
	iStateStoping							: INT;
	iStateAborting							: INT;	
	fbPower 								:MC_Power;
	fbMove	 								:MC_MoveAbsolute;
	fbJog 									:MC_Jog;
	fbReset 								:MC_Reset;	
	fbStop									:MC_Stop;
	//fbBeltInverter							:FB_MX2;
	arrErrorTable							:ARRAY[0..1000] OF UDINT;
	arrError								:ARRAY[0..1000] OF BOOL;
	tonAxesReady							:TON;
	tonAxesError							:TON;
	fbBeltInverter							:FB_INV003_MX2_ECT;
END_VAR
(*----------------------------------------------Koniec nowego dopisanego -------------------------------*)

ACTION Ack_FBsCall:
//Servo Axis Fb`s
	
fbPower(
	Axis:=GVL_AXIS.stAxis1 , 
	Enable:=, 
	Enable_Positive:=GVL_AXIS.bEnable , 
	Enable_Negative:=GVL_AXIS.bEnable , 
	Override:=100.0 , 
	BufferMode:= , 
	Options:= , 
	Status=> , 
	Busy=> , 
	Active=> , 
	Error=> arrError[0], 
	ErrorID=>arrErrorTable[0] );

fbReset(
	Axis:= GVL_AXIS.stAxis1, 
	Execute:= , 
	Done=> , 
	Busy=> , 
	Error=>	arrError[1] , 
	ErrorID=>arrErrorTable[1] );
		
fbJog(
	Axis:= GVL_AXIS.stAxis1, 
	JogForward:= bJog_B , 
	JogBackwards:=bJog_F , 
	Mode:= , 
	Position:= , 
	Velocity:= GVL_HMI.J_VelK, 
	Acceleration:= , 
	Deceleration:= , 
	Jerk:= , 
	Done=> , 
	Busy=> , 
	Active=> , 
	CommandAborted=> , 
	Error=> arrError[2] , 
	ErrorID=>arrErrorTable[2] );
	
fbMove(
	Axis:=GVL_AXIS.stAxis1 , 
	Execute:= bExecute, 
	Position:=Position , 
	Velocity:=Predkosc , 
	Acceleration:= , 
	Deceleration:= , 
	Jerk:= , 
	BufferMode:= , 
	Options:= , 
	Done=> , 
	Busy=> , 
	Active=> , 
	CommandAborted=> , 
	Error=>arrError[3] , 
	ErrorID=>arrErrorTable[3]
 );
 fbStop(
	Axis:=GVL_AXIS.stAxis1 , 
	Execute:= , 
	Deceleration:= , 
	Jerk:= , 
	Options:= , 
	Done=> , 
	Busy=> , 
	Active=> , 
	CommandAborted=> , 
	Error=> arrError[4] , 
	ErrorID=>arrErrorTable[4] );
	//Inverters fb`s nie używany 
(*fbBeltInverter
	(w_Status:=GVL_Omron.wOmron_1_Status,
	ui_CzestotliwoscI:=F1_FQ,
	b_CCW:=F1_CW, 
	b_CW:=F1_CCW, 
	b_Reset:=F_Reset,		
	w_ControlW=>GVL_Omron.wOmron_1_Control,
 	ui_CzestotliwoscO=>GVL_Omron.iOmron_1_SeVelo,);
*)	
(*
fbBeltInverter(
	Output_Frequency_Monitor:=GVL_Omron.iOmron_1_ActVelo , 
	During_Rev:= , 
	Enable:= , 
	Fwd:= , 
	Rev:= , 
	Fault_Reset:= , 
	Frequency_in:= , 
	Acceleration:= , 
	Deceleration:= , 
	ENO=> , 
	Frequency_out=>GVL_Omron.iOmron_1_SeVelo , 
	During_Fwd=> , 
	Fault=>arrError[5], 
	Warning=> , 
	Remote=> , 
	Freq_Match=> , 
	Connection_Error=> , 
	Command:=GVL_Omron.wOmron_1_Status , 
	Frequency_Reference:= , 
	F002_1st_Acceleration:=GVL_Omron.iOmronErectorAcc , 
	F003_1st_Deceleration:=GVL_Omron.iOmronErectorDcc , 
	Status:=GVL_Omron.wOmron_1_Status);
*)
END_ACTION

ACTION Ack_IOLinkRequest:
//załączenie kanału io-link Kanał 1 
		GVL_IO.IOLinkCh1T:=TRUE;
END_ACTION

ACTION Act_ButtonsLight:
IF  (gvl_hmi.A_Start=TRUE  THEN GVL_IO.K1K5:=FALSE; GVL_IO.K1K7:=TRUE; ; END_IF
IF gvl_hmi.A_Stop=TRUE THEN GVL_IO.K1K5:=TRUE; GVL_IO.K1K7:=FALSE;  END_IF
GVL_HMI.A_Start:=gvl_Io.b1K1;
GVL_HMI.A_Stop:=GVL_IO.b1K3;
END_ACTION

ACTION Act_Error:

END_ACTION

ACTION Act_Magazine:
K_Magazyn(
	bStop:=GVL_IO.b1K3 AND GVL_HMI.bAuto,
	xPodjedz:=GVL_IO.b1K1, 
	xWydajKarton:=, 
	xKartonPobrany:=, 
	xCzPodjazd:=, 
	xCzTrzymacz2:=, 
	xCzTrzymacz1:=GVL_IO.bCzujnik_Trzymacz1, 
	xSilPodpych=>GVL_IO.K1K4, 
	xSilTrzymacz1=>GVL_IO.K1K1, 
	xSilTrzymacz2=>GVL_IO.K1K3, 
	xWydalemKarton=>, 
	xBlad=> );
END_ACTION

ACTION Act_ModeAutomatic:
// State Machine
(*
CASE eMachineState OF

	E_MachineState.eIdle:
		
	
		// ====================================================
		// There should be main code
		// i.e. CASE iStepInit OF	
		// ====================================================
		// Allow for stop only if conditions are true - in this step we can wait without an error

		
		IF TRUE (* condition *) THEN
			eMachineState 						:= E_MachineState.eStopped;
		END_IF
		
		IF bError THEN
			eMachineState 						:= E_MachineState.eError;
		END_IF
		
	E_MachineState.eStopping:
		
		
		CASE iStateStoping OF
			0:
				
			
			10:
			
			20:
				
		END_CASE
		IF iStateStoping = 20 (* condition *) THEN
			eMachineState 						:= E_MachineState.eStopped;
			iStateStoping 						:= 0;
		END_IF		
	
	E_MachineState.eStopped:
		
	
		
		IF eMachineCommand = E_MachineCommand.eRun THEN
			eMachineState 						:= E_MachineState.eStarting;
		END_IF
		
		IF eMachineCommand = E_MachineCommand.eRestart THEN
			GVL_MachineMaintenance.eCommand		:= E_MachineCommand.eStop;
			eMachineState 						:= E_MachineState.eRestarting;
		END_IF			
				
		IF bError THEN
			eMachineState 						:= E_MachineState.eError;
		END_IF

	E_MachineState.eStarting:
	

		CASE iStepStarting OF
			0:		
				fbPower.Enable:=TRUE;
				
				IF tonAxesReady.Q THEN
					iStepStarting := iStepStarting + 10;
				ELSIF tonAxesError.Q THEN
					bError := TRUE;
				END_IF
			
			10:
			
				IF (*Warunki startu automatu*)  THEN
					iStepStarting := iStepStarting + 20;		
				ELSE
					bError := TRUE;
					iStepStarting := iStepStarting + 10;
				END_IF
				
			20:
			
		
				
			END_CASE 
	
		IF iStepStarting = 20 AND (*Kartoniarka READY*) THEN
			eMachineState 						:= E_MachineState.eRunning;
			iStepStarting 						:= 0;
		END_IF
		
			
		
	E_MachineState.eRunning:
		

		// ====================================================
		// There should be main code
		// i.e. CASE iStepAuto OF
		// ====================================================
		IF eMachineCommand = E_MachineCommand.eStop OR bError THEN
			eMachineState 						:= E_MachineState.eStopping;
		END_IF

	E_MachineState.eAborting:

		// Stop and reset everything - usually SAFETY function
		CASE iStateAborting OF
			0:
				IF (*warunek wykonania zatrzymania *) THEN
					iStateAborting := iStateAborting +10;
				END_IF
			10:
				
						fbMove.Execute:= FALSE;
						fbStop.Execute:= FALSE;
						
						IF fbStop.Done THEN
							iStateAborting := iStateAborting +10;	
						END_IF
				
			20:
						fbPower.Enable:=FALSE;
					IF NOT fbPower.Status THEN 
						iStateAborting := iStateAborting + 10;
					END_IF
			30:
			
					
				
		END_CASE
	
		IF iStateAborting = 30 THEN
			eMachineState 						:= E_MachineState.eAborted;
			iStateAborting						:= 0;
		END_IF		
		
	E_MachineState.eAborted:

					
		IF eMachineCommand = E_MachineCommand.eReset THEN
			eMachineState 						:= E_MachineState.eReseting;
		END_IF
		
		IF bError THEN
			eMachineState 						:= E_MachineState.eError;
		END_IF

	E_MachineState.eError:

		// ====================================================
		// Two types of error:
		// 1. 'Small/soft' Error - fix a problem and go to stop
		// 2. 'Serious/hard' Error - there is a need of restart everything, if there is a sequence - reset it too - fix a problem and go to init
		// ====================================================

	
	
		IF eMachineCommand = E_MachineCommand.eReset THEN
			eMachineState 						:= E_MachineState.eReseting;
		END_IF
		
		IF eMachineCommand = E_MachineCommand.eRestart THEN
			eMachineState 						:= E_MachineState.eRestarting;
		END_IF

	E_MachineState.eReseting:

		// ====================================================
		//'Small/soft' Error - fix a problem and go to stop
		// Reset drives only when it is necessary
		// ====================================================
		// Check if axis errors cleared
	
		IF fbPower.Error	THEN
			fbReset.Execute := TRUE;
		ELSIF fbBeltInverter.Fault THEN
			fbBeltInverter.Fault_Reset:=TRUE;
		END_IF

	
		IF NOT tonAxesError.Q  THEN
			fbReset.Execute := FALSE;
			fbBeltInverter.Fault_Reset:=FALSE;
		END_IF
				
		// Blad bloku resetowania lub zakonczylismy kasowanie bledu osi, ale os jest nadal w bledzie, np. nie usunieta usterka - idz do kroku bledu
		IF bError (*(stAxis.stAxisDiagOutputs.Error OR (stAxis.stAxisDiagOutputs.Done AND stAxis.bAxisError)) *) THEN
			eMachineState  						:= E_MachineState.eError;
		END_IF
		
	E_MachineState.eRestarting:

		// ====================================================
		// 'Serious/hard' Error - there is a need of restart everything, if there is a sequence - reset it too - fix a problem and go to init
		// Reset drives only when it is necessary
		// ====================================================
		// Check if axis errors cleared
		bError := FALSE;
		
		IF TRUE (*NOT bAxisError AND NOT other errors *) THEN
			eMachineState  						:= E_MachineState.eIdle;
		END_IF
				
		// Blad bloku resetowania lub zakonczylismy kasowanie bledu osi, ale os jest nadal w bledzie, np. nie usunieta usterka - idz do kroku bledu
		IF bError (*(stAxis.stAxisDiagOutputs.Error OR (stAxis.stAxisDiagOutputs.Done AND stAxis.bAxisError)) *) THEN
			eMachineState  						:= E_MachineState.eError;
		END_IF
		
END_CASE
*)
END_ACTION

ACTION Act_ModeManual:

END_ACTION

ACTION Act_Monitoring:
tonAxesReady(PT:=T#200MS);
tonAxesReady.IN:=fbPower.Active;

tonAxesError(PT:=T#200MS);
tonAxesError.IN:=arrError[0] OR arrError[1] OR arrError[2]  OR arrError[5]
							 OR arrError[3] OR arrError[4];
END_ACTION

END_PROGRAM

// ---- POUs/Programy/PRG_CaseMachineMode.TcPOU
PROGRAM PRG_CaseMachineMode
VAR
	//	GVL_Machine - HMI handling
	bHMIModeRequest_Automatic			: BOOL;
	bHMIModeRequest_Manual				: BOOL;
	
	bHMICommandRequest_Run				: BOOL;
	bHMICommandRequest_Stop				: BOOL;
	bHMICommandRequest_Reset			: BOOL;
	bHMICommandRequest_Restart			: BOOL;
	bHMICommandRequest_Abort			: BOOL;
	
	// Rising edge detection
	rtButtonAutomatic					: R_TRIG;
	rtButtonManual						: R_TRIG;
	rtButtonMaintenance					: R_TRIG;
	rtButtonStart						: R_TRIG;
	rtButtonReset						: R_TRIG;
	rtButtonStop						: R_TRIG;
	// State change permissions
	bAllowChangeToManual				: BOOL;
	bAllowChangeToMaintenance			: BOOL;
	bAllowChangeToAutomatic				: BOOL;
	rtButtonEnable: R_TRIG;
	bHMICommandRequest_Enable: BOOL;
END_VAR

// Triggers
rtButtonAutomatic(CLK:= bHMIModeRequest_Automatic );
rtButtonManual(CLK:= bHMIModeRequest_Manual );
rtButtonStart(CLK:= bHMICommandRequest_Run);
rtButtonStop(CLK:= bHMICommandRequest_Stop);
rtButtonReset(CLK:= bHMICommandRequest_Reset);


//przepisanie zmiennych
bHMICommandRequest_Run										:= GVL_IO.B1K1;
bHMICommandRequest_Stop										:= GVL_IO.B1K3;
bHMICommandRequest_Reset									:= GVL_IO.B1K8;
bHMIModeRequest_Automatic									:= GVL_IO.di_Auto;
bHMICommandRequest_Enable									:= GVL_HMI.bEnableKartoniarka;

// SAFETY niezaleznie
IF NOT GVL_SafetyFrom_RT2.bSAFETY_PermissionSS1 OR bHMICommandRequest_Abort THEN
	GVL_MachineMaintenance.eCommand							:= E_MachineCommand.eAbort;
	GVL_MachineMaintenance.eState							:= E_MachineState.eAborted;
END_IF

//uruchomienie automatu 


// przełączynik trybu auto/manual
IF GVL_HMI.bAuto THEN
	bHMIModeRequest_Automatic 								:= TRUE;
	bHMIModeRequest_Manual 									:= FALSE;
ELSE
	bHMIModeRequest_Automatic 								:= FALSE;
	bHMIModeRequest_Manual 									:= TRUE;
END_IF

CASE GVL_MachineMaintenance.eMode OF 

	E_MachineMode.eAutomatic:

		// Zmiana trybu tylko gdy maszyna nie jest w Running
		IF GVL_MachineMaintenance.eState <> E_MachineState.eRunning THEN
			IF rtButtonMaintenance.Q THEN
				GVL_Machine.eCommand						:= E_MachineCommand.eRestart;
				GVL_Machine.eMode							:= E_MachineMode.eMaintenance;
			END_IF
		END_IF
		
		IF GVL_MachineMaintenance.eState <> E_MachineState.eRunning THEN
			IF rtButtonManual.Q THEN
				GVL_MachineMaintenance.eCommand				:= E_MachineCommand.eRestart;
				GVL_MachineMaintenance.eMode				:= E_MachineMode.eManual;
			END_IF
		END_IF
		//==============================================
		IF rtButtonStart.Q THEN 
			GVL_MachineMaintenance.eCommand					:= E_MachineCommand.eRun;
		END_IF

		IF rtButtonReset.Q AND GVL.bRestartRequired THEN
			GVL_MachineMaintenance.eCommand					:= E_MachineCommand.eRestart;
		END_IF
		
		IF rtButtonReset.Q AND NOT GVL.bRestartRequired THEN
			GVL_MachineMaintenance.eCommand					:= E_MachineCommand.eReset;
		END_IF
		
		IF GVL.bGeneralError OR GVL.bGeneralFatalError OR rtButtonStop.Q THEN
			GVL_MachineMaintenance.eCommand					:= E_MachineCommand.eStop ;
		END_IF
		
	E_MachineMode.eMaintenance, E_MachineMode.eManual:
	
		// Reset, Restart, Error - not used
		
		// Zmiana trybu tylko gdy maszyna nie jest w Running
		IF GVL_MachineMaintenance.eState <> E_MachineState.eRunning  THEN
			IF rtButtonAutomatic.Q AND bHMICommandRequest_Enable THEN
				GVL_MachineMaintenance.eCommand				:= E_MachineCommand.eRestart;
				GVL_MachineMaintenance.eMode				:= E_MachineMode.eAutomatic;
			END_IF
		END_IF
		
		//==============================================
		IF rtButtonStart.Q THEN 
			GVL_MachineMaintenance.eCommand 				:= E_MachineCommand.eRun;
		END_IF

		IF rtButtonReset.Q AND GVL.bRestartRequired THEN
			GVL_MachineMaintenance.eCommand					:= E_MachineCommand.eRestart;
		END_IF
		
		IF rtButtonReset.Q AND NOT GVL.bRestartRequired THEN
			GVL_MachineMaintenance.eCommand					:= E_MachineCommand.eReset;
		END_IF
		
		IF rtButtonStop.Q THEN
			GVL_MachineMaintenance.eCommand					:= E_MachineCommand.eStop ;
		END_IF

END_CASE

END_PROGRAM

// ---- VISUs/GlobalTextList.TcGTLO
TEXTLIST GlobalTextList
  116 = '   Actual Velocity [mm/s]:'
  115 = '   Error:'
  282 = '   Position [mm]:'
  112 = '   Setpoint Position [mm]:'
  114 = '   Setpoint Velocity [mm/s]:'
  1684 = ' a następnie"Create recipe"'
  1317 = '!'
  1322 = '"'
  2204 = '#'
  1327 = '$'
  1333 = '%'
  120 = '%.2f'
  281 = '%.4f'
  279 = '%3.0f'
  256 = '%3.1f'
  259 = '%3.2f'
  1817 = '%d'
  551 = '%f'
  273 = '%i'
  318 = '%s'
  762 = '%S'
  204 = '%s 4'
  976 = '%sl'
  1338 = '&'
  210 = "'"
  1343 = '('
  924 = ')'
  1301 = '*'
  474 = '+'
  475 = '+ +'
  211 = ','
  476 = '-'
  477 = '- -'
  212 = '.'
  214 = '/'
  1954 = '0'
  942 = '1'
  1585 = '1. Create recipe'
  784 = '1. Naciśnij "Create recipe"'
  2669 = '1. Naciśnij wolny wiersz w tabeli "Recepty",'
  261 = '1. Naciśnij wolny wiersz w tabeli "Recepty", a następnie"Create recipe"'
  946 = '2'
  2172 = '2. Naciśnij " Save as"'
  2602 = '2. Wprowadź wartości'
  950 = '3'
  2925 = '3. Naciśnij " Save values"'
  3229 = '3. Wprowadź wartości do tabeli'
  953 = '4'
  2363 = '4. Naciśnij " LOAD"'
  733 = '4. Naciśnij " Save values"'
  1059 = '4. Naciśnij " Save"'
  1700 = '4. Naciśnij "Load Recipe"'
  2070 = '4. Naciśnij "Load"'
  1918 = '5'
  974 = '5. Naciśnij " Save as"'
  262 = '5. Naciśnij "Load Recipe"'
  639 = '5. Naciśnij "Save recipe"'
  1925 = '6'
  398 = '6. Naciśnij "Save recipe"'
  1932 = '7'
  1940 = '8'
  1947 = '9'
  1264 = ':'
  209 = ';'
  1481 = '<'
  1961 = '='
  1489 = '>'
  928 = '?'
  2213 = '@'
  1276 = 'a'
  1282 = 'A'
  726 = 'Aktualne wartości PLC'
  760 = 'Alarmy'
  469 = 'All'
  1123 = 'AUTOMAT'
  555 = 'Axis Error ?'
  272 = 'Axis ID'
  274 = 'Axis Name'
  1229 = 'b'
  1234 = 'B'
  1450 = 'Backspace'
  647 = 'Bezpieczeństwo OK'
  268 = 'Błąd'
  985 = 'Błąd kartoniarka'
  628 = 'Błąd kierownica'
  1033 = 'Błędy'
  1203 = 'c'
  1209 = 'C'
  288 = 'Calibrated'
  1443 = 'Clear'
  276 = 'Controller'
  284 = 'Coupled Mode'
  841 = 'Create recipe'
  845 = 'Current PLC values'
  852 = 'Current recipe definiton:'
  853 = 'Current recipe:'
  1228 = 'Czujnik hamulec'
  1167 = 'Czujnik hamulec 1'
  1394 = 'Czujnik hamulec 2'
  1196 = 'Czujnik obecności taśmy'
  8 = 'Czujnik prawidło dół'
  1139 = 'Czujnik prawidło góra'
  407 = 'Czujnik siłownika zamykacza'
  775 = 'Częstotliwość'
  1442 = 'Częstotliwość Aktualna'
  1300 = 'd'
  1307 = 'D'
  2968 = 'Dane recepty'
  844 = 'Delete recipe'
  92 = 'Diagnostyka'
  133 = 'Dojki'
  847 = 'DWORD value:'
  1907 = 'Długość kartonu:'
  2262 = 'e'
  1887 = 'E'
  139 = 'EnableAxes'
  297 = 'EnableKinAxes'
  643 = 'EnableKinematic'
  275 = 'Enabling'
  1435 = 'ESC'
  1313 = 'f'
  1319 = 'F'
  788 = 'Falownik pasów'
  1434 = 'Falownik podajnik'
  1437 = 'Falownik rolek'
  277 = 'Feed Bw'
  278 = 'Feed Fw'
  616 = 'Force Lock'
  617 = 'Force Unlock'
  1325 = 'g'
  1331 = 'G'
  1065 = 'Gotowa'
  824 = 'GroupBox'
  2126 = 'h'
  2136 = 'H'
  290 = 'Has Job'
  478 = 'HBOT Os X'
  522 = 'HBOT Os Y'
  471 = 'HOME'
  1959 = 'i'
  1967 = 'I'
  615 = 'I2T Max [%]:'
  614 = 'I2T [%]:'
  124 = 'Ilość kolumn:'
  3000 = 'Ilość rzędów'
  286 = 'In Position Range'
  285 = 'In Target Position'
  351 = 'Informacje'
  846 = 'INT value:'
  2146 = 'j'
  2155 = 'J'
  1573 = 'Jog +'
  2205 = 'Jog -'
  2165 = 'k'
  2175 = 'K'
  315 = 'Kartoniarka'
  138 = 'Kartoniarka  '
  121 = 'Kartoniarka Ready'
  473 = 'Kierownica'
  681 = 'Kinematyka OK'
  539 = 'Kinematyka Ploter OK'
  189 = 'Klapka długa schowana'
  1467 = 'Klapka długa wysunięta'
  350 = 'Klapka krótka schowana'
  871 = 'Klapka krótka wysunięta'
  1035 = 'Klapka schowana'
  263 = 'Kolejny'
  2184 = 'l'
  2194 = 'L'
  117 = 'Lag Distance [mm]:'
  854 = 'Last error (0 == OK):'
  930 = 'Liczba recept'
  205 = 'List of existing recipes for the current recipe definiton:'
  505 = 'Listar zapisanych recept'
  840 = 'Load recipe'
  843 = 'Load recipe from'
  1252 = 'm'
  1259 = 'M'
  626 = 'Magazyn +'
  857 = 'Magazyn -'
  935 = 'Max:'
  932 = 'Min:'
  110 = 'Moving Bw'
  109 = 'Moving Fw'
  1240 = 'n'
  1246 = 'N'
  856 = 'Name'
  199 = "Name and value of the current recipe's variables:"
  190 = 'Nazwa i wartości aktualnej recepty'
  2846 = 'Nazwa recepty'
  2542 = 'Nazwa Recepty'
  715 = 'Nazwy i wartości zmiennych'
  849 = 'New recipe name:'
  108 = 'NOT Moving'
  2334 = 'Nowe wartości'
  1125 = 'Nr błędu'
  1064 = 'Nr błędu:'
  1975 = 'o'
  1983 = 'O'
  87 = 'Obecna definicja:'
  595 = 'Obecna recepta'
  869 = 'Obecne wartości'
  1530 = 'Obecne wartości '
  1427 = 'OK'
  2080 = 'ON'
  949 = 'ON/OFF'
  934 = 'Os X'
  47 = 'Os Y'
  1777 = 'Ostatni błąd (0 == OK):'
  280 = 'Override [%]'
  118 = 'Override [%]:'
  1991 = 'p'
  1999 = 'P'
  1084 = 'Panel komend'
  632 = 'Pauza'
  228 = 'Ploter'
  1094 = 'Ploter Ready'
  1 = 'Pobranie'
  172 = 'Podajnik Ready'
  173 = 'Pozycja głowicy kartoniarki'
  583 = 'Pozycja kierownicy'
  1081 = 'Pozycja magazynu kartonów'
  1458 = 'Pozycja serwa'
  1762 = 'Pozycja X odłożenia:'
  1077 = 'Pracuje'
  777 = 'Prędkość Serwo mm/s'
  2223 = 'q'
  2233 = 'Q'
  1895 = 'r'
  1903 = 'R'
  838 = 'Read variables into recipe'
  111 = 'Ready'
  848 = 'REAL value:'
  35 = 'Recepty'
  480 = 'Recipe commands'
  855 = 'Recipe count:'
  851 = 'Recipe information'
  850 = 'Recipe Management'
  1743 = 'Recipe Mnagement'
  203 = 'Recipes'
  119 = 'Ref Velo [mm/s]:'
  207 = 'Refresh'
  289 = 'Reset'
  472 = 'RESET'
  1565 = 'Reset Błędu'
  255 = 'Reset Max'
  1288 = 's'
  1294 = 'S'
  201 = 'Save'
  839 = 'Save recipe'
  842 = 'Save recipe as'
  2752 = 'Save Values'
  36 = 'SelectionIndex: %s'
  6 = 'Serwis'
  576 = 'Serwo '
  1291 = 'Serwo Error'
  421 = 'Serwo Jog+'
  535 = 'Serwo Jog-'
  761 = 'Serwo Ready'
  1459 = 'Shift'
  479 = 'Sieć'
  482 = 'Siłownik zamykacz'
  1992 = 'Skos'
  1465 = 'Space'
  541 = 'START'
  113 = 'Start'
  287 = 'Status (log.)'
  283 = 'Status (phys.)'
  213 = 'Status Maszyny'
  305 = 'STATUSY'
  37 = 'Statusy'
  564 = 'Statystyki'
  470 = 'STOP'
  331 = 'Stop'
  423 = 'Szerokość kartonu:'
  1911 = 't'
  1919 = 'T'
  467 = 'Target Pos [mm]:'
  468 = 'Target Velo [mm/s]:'
  592 = 'Taśmy'
  258 = 'Torque Error'
  260 = 'Torque Filter[Nm]:'
  257 = 'Torque Limit [%]:'
  619 = 'Torque Max [%]:'
  613 = 'Torque Max [Nm]:'
  618 = 'Torque [%]:'
  291 = 'TWORZĄC NOWĄ RECEPTĘ'
  1943 = 'u'
  1951 = 'U'
  441 = 'UWAGA !!! '
  938 = 'UWAGA !!! TWORZENIE NOWEJ RECEPTY '
  1215 = 'v'
  1221 = 'V'
  197 = 'Value'
  2242 = 'w'
  2252 = 'W'
  552 = 'Wartość'
  481 = 'Write recipe into variables'
  368 = 'Wróć'
  122 = 'Wybrany numer recepty: %s'
  793 = 'Wydajność'
  544 = 'Wydajność '
  310 = 'Wymuś pobranie'
  104 = 'Wypychacz przód'
  157 = 'Wypychacz tył'
  1395 = 'Wysokość kartonu:'
  1512 = 'x'
  1197 = 'X'
  1496 = 'y'
  1504 = 'Y'
  1927 = 'z'
  1935 = 'Z'
  585 = 'Zaklejarka'
  969 = 'Zaklejarka Ready'
  1258 = 'Zakręcarka'
  1764 = 'Zaladuj'
  566 = 'Zawór chwytaka 1'
  1013 = 'Zawór chwytaka 2'
  1206 = 'Zawór hamulec '
  557 = 'Zawór hamulec 1'
  895 = 'Zawór hamulec 2'
  1306 = 'zawór klapki długie'
  1060 = 'Zawór klapki długie'
  1617 = 'zawór klapki krótkie'
  412 = 'Zawór klapki krótkie'
  610 = 'Zawór prawidło'
  620 = 'Zawór prawidło dół'
  778 = 'Zawór ssawki'
  687 = 'Zawór wypychacz'
  2455 = 'Załadował'
  177 = 'zz'
  1860 = 'Zęby'
  1976 = '['
  1997 = '\\'
  1990 = ']'
  1312 = '^'
  1270 = '_'
  1968 = '{'
  1473 = '|'
  1984 = '}'
  1308 = '~'
  939 = '´'
END_TEXTLIST

// ---- VISUs/Glowna.TcVIS
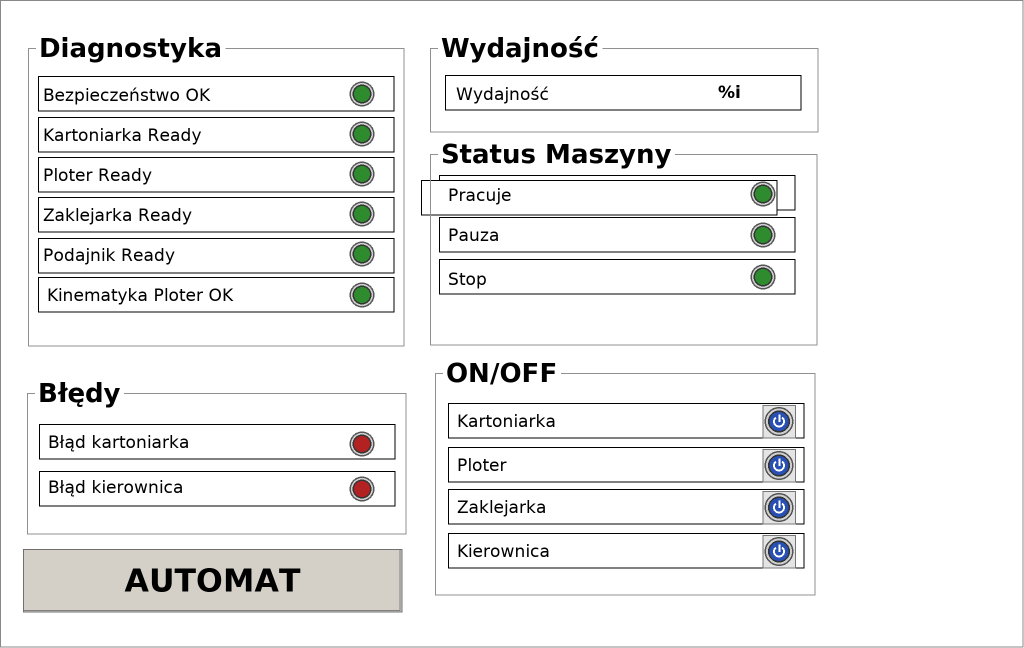
VISUALIZATION Glowna  // 1024x648
    Rectangle (439,175 356x35)
    GroupBox (28,40 376x306), "Diagnostyka"
        Rectangle (10,198 356x35)
        Rectangle (10,157 356x35)
        Rectangle (10,117 356x35)
        Rectangle (10,77 356x35)
        Rectangle (10,36 356x35)
        Label (12,40 209x30), "Bezpieczeństwo OK"
        Label (12,80 209x30), "Kartoniarka Ready"
        Label (12,160 209x30), "Zaklejarka Ready"
        Label (12,200 209x30), "Podajnik Ready"
        Lamp1 (320,40 28x28), variable: GVL_SafetyFrom_RT2.bSAFETY_PermissionSS1 and GVL_SafetyFrom_RT2.bSAFETY_PermissionSS2, style: Lamp-Lamp1-Green
        Lamp1 (320,80 28x28), style: Lamp-Lamp1-Green
        Lamp1 (320,120 28x28), style: Lamp-Lamp1-Green
        Lamp1 (320,200 28x28), style: Lamp-Lamp1-Green
        Lamp1 (320,160 28x28), style: Lamp-Lamp1-Green
        Rectangle (10,237 356x35)
        Label (16,240 209x30), "Kinematyka Ploter OK"
        Lamp1 (320,241 28x28), style: Lamp-Lamp1-Green
        Label (12,120 209x30), "Ploter Ready"
        Rectangle (393,140 356x35)
    GroupBox (430,40 388x92), "Wydajność"
        Rectangle (15,35 356x35)
        Label (23,39 209x30), "Wydajność"
        Label (209,101 100x25)
        Textfield (239,37 121x30), "%i", text variable: GVL_HMI.iWydajnosc
    GroupBox (435,365 380x230), "ON/OFF"
        Rectangle (13,38 356x35)
        Label (19,41 209x30), "Kartoniarka"
        Rectangle (13,82 356x35)
        Label (19,85 209x30), "Ploter"
        Rectangle (13,168 356x35)
        Label (19,171 209x30), "Kierownica"
        Rectangle (13,124 356x35)
        Label (19,127 209x30), "Zaklejarka"
        PowerSwitch (325,40 38x33), variable: GVL_HMI.bEnableKartoniarka, behaviour: TOGGLE, style: Switch-PowerSwitch-Blue
        PowerSwitch (325,84 38x33), variable: GVL_HMI.bEnablePloter, behaviour: TOGGLE, style: Switch-PowerSwitch-Blue
        PowerSwitch (325,126 38x33), variable: GVL_HMI.bEnableZaklejarka, behaviour: TOGGLE, style: Switch-PowerSwitch-Blue
        PowerSwitch (325,170 38x33), variable: GVL_HMI.bEnableKierownica, behaviour: TOGGLE, style: Switch-PowerSwitch-Blue
    GroupBox (430,146 387x199), "Status Maszyny"
        Label (211,97 100x25)
    Label (445,180 209x30), "Pracuje"
    Lamp1 (749,180 28x28), style: Lamp-Lamp1-Green
    Rectangle (439,217 356x35)
    Label (445,220 209x30), "Pauza"
    Lamp1 (749,221 28x28), style: Lamp-Lamp1-Green
    Rectangle (439,259 356x35)
    Label (445,264 209x30), "Stop"
    Lamp1 (749,263 28x28), style: Lamp-Lamp1-Green
    GroupBox (27,385 379x149), "Błędy"
        Textfield (240,41 121x30), text variable: GVL_HMI.INT_idError
        Rectangle (12,39 356x35)
        Label (18,42 209x30), "Błąd kartoniarka"
        Lamp1 (321,45 28x28), variable: GVL_GLOBAL.Error_ind_kart, style: Lamp-Lamp1-Red
        Rectangle (12,86 356x35)
        Lamp1 (321,90 28x28), variable: GVL_GLOBAL.Error_pakowania, style: Lamp-Lamp1-Red
        Label (18,87 209x30), "Błąd kierownica"
    Button (23,549 379x63), "AUTOMAT"
        toggle GVL_HMI.bAutoWybor
END_VISUALIZATION

// ---- VISUs/HMI.TcVIS
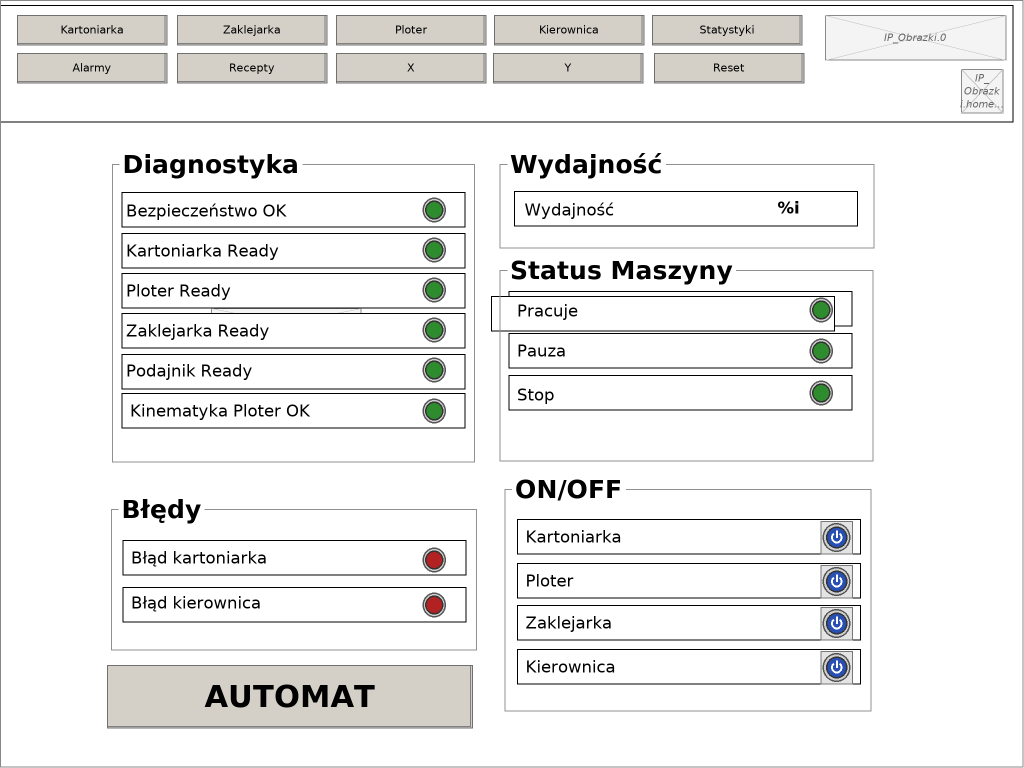
VISUALIZATION HMI  // 1024x768
    Rectangle (-1,5 1014x117)
    Button (17,15 150x30), "Kartoniarka", colour toggle: GVL_HMI.strona=1
        OnMouseDown: FrameSelectionChange Selection=SelectedFrame=f7e3fd18-cbcb-49a2-8593-590d8a027e7f, Selection=1, GlobSel=AssignType=Directly, SelType=Locally
        OnMouseDown: execute { gvl_hmi.strona:=1; }
    Button (177,15 150x30), "Zaklejarka", colour toggle: GVL_HMI.strona=2
        OnMouseDown: FrameSelectionChange Selection=SelectedFrame=f7e3fd18-cbcb-49a2-8593-590d8a027e7f, Selection=7, GlobSel=AssignType=Directly, SelType=Locally
        OnMouseDown: execute { gvl_hmi.strona:=2; }
    Button (654,53 150x30), "Reset", colour toggle: GVL_SafetyFrom_RT2.bSAFETY_PermissionSS1=true and GVL_SafetyFrom_RT2.bSAFETY_PermissionSS2=true
        tap GVL_SafetyFrom_RT2.bSAFETY_ResetCMD
    Button (336,15 150x30), "Ploter", colour toggle: GVL_HMI.strona=3
        OnMouseDown: execute { gvl_hmi.strona:=3; }
        OnMouseDown: FrameSelectionChange Selection=SelectedFrame=f7e3fd18-cbcb-49a2-8593-590d8a027e7f, Selection=3, GlobSel=AssignType=Directly, SelType=Locally
    Button (494,15 150x30), "Kierownica", colour toggle: GVL_HMI.strona=4
        OnMouseDown: execute { gvl_hmi.strona:=4; }
        OnMouseDown: FrameSelectionChange Selection=SelectedFrame=f7e3fd18-cbcb-49a2-8593-590d8a027e7f, Selection=2, GlobSel=AssignType=Directly, SelType=Locally
    Image (825,15 181x45), image: IP_Obrazki.0
    Button (177,53 150x30), "Recepty", colour toggle: GVL_HMI.strona=6
        OnMouseDown: FrameSelectionChange Selection=SelectedFrame=f7e3fd18-cbcb-49a2-8593-590d8a027e7f, Selection=6, GlobSel=AssignType=Directly, SelType=Locally
        OnMouseDown: execute { gvl_hmi.strona:=6; }
    Button (336,53 150x30), "X", colour toggle: GVL_HMI.strona=22
        OnMouseDown: FrameSelectionChange Selection=SelectedFrame=f7e3fd18-cbcb-49a2-8593-590d8a027e7f, Selection=9, GlobSel=AssignType=Directly, SelType=Locally
        OnMouseDown: execute { gvl_hmi.strona:=22; }
    Button (17,53 150x30), "Alarmy", colour toggle: GVL_HMI.strona=5
        OnMouseDown: execute { gvl_hmi.strona:=5; }
        OnMouseDown: FrameSelectionChange Selection=SelectedFrame=f7e3fd18-cbcb-49a2-8593-590d8a027e7f, Selection=8, GlobSel=AssignType=Directly, SelType=Locally
    ImageSwitcher (211,308 150x30), behaviour: TOGGLE
    Image (961,69 42x44), colour toggle: GVL_HMI.strona=0, image: IP_Obrazki.home-icon-silhouette (1)
        OnMouseDown: FrameSelectionChange Selection=SelectedFrame=f7e3fd18-cbcb-49a2-8593-590d8a027e7f, GlobSel=AssignType=Directly, SelType=Locally
        OnMouseDown: execute { gvl_hmi.strona:=0; }
    Button (652,15 150x30), "Statystyki", colour toggle: GVL_HMI.strona=8
        OnMouseDown: execute { gvl_hmi.strona:=8; }
        OnMouseDown: FrameSelectionChange Selection=SelectedFrame=f7e3fd18-cbcb-49a2-8593-590d8a027e7f, Selection=5, GlobSel=AssignType=Directly, SelType=Locally
    Button (493,53 150x30), "Y", colour toggle: GVL_HMI.strona=7
        OnMouseDown: FrameSelectionChange Selection=SelectedFrame=f7e3fd18-cbcb-49a2-8593-590d8a027e7f, Selection=10, GlobSel=AssignType=Directly, SelType=Locally
        OnMouseDown: execute { gvl_hmi.strona:=7; }
    Frame (85,116 988x648)
        shows Glowna()
        shows Kartoniarka()
        shows Kierwonica()
        shows Ploter()
        shows Serwis()
        shows Statystyki()
        shows Visualization()
        shows Zaklejarka()
        shows Alarmy()
        shows PH_AxisOnline(stMcAxisOnline := P_HBot_v3.stMcAxisOnline_MCS_X)
        shows PH_AxisOnline_1(stMcAxisOnline := P_HBot_v3.stMcAxisOnline_MCS_Y)
END_VISUALIZATION

// ---- VISUs/Alarmy.TcVIS
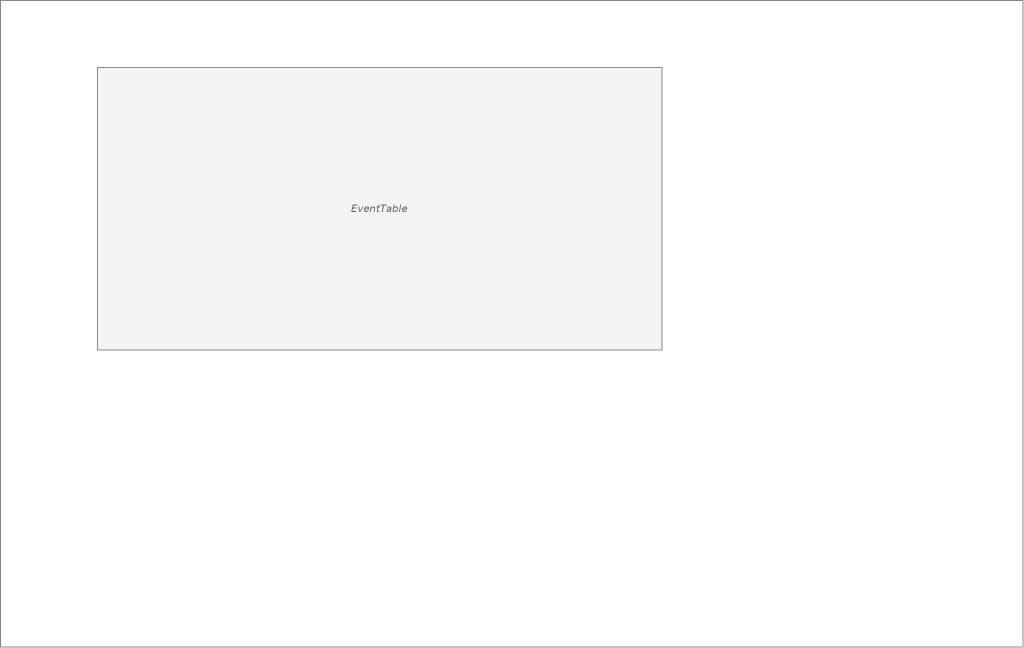
VISUALIZATION Alarmy  // 1024x648
    EventTable (97,67 565x283)
        p1690906150: Class
        p3258520714: Date
        p2231227367: Time
        p3993844394: Message
        p2076579579: Details
        p3558512729: aEventsSimple
        p3921149237: m_pDataArray..pArray
END_VISUALIZATION

// ---- VISUs/Kartoniarka.TcVIS
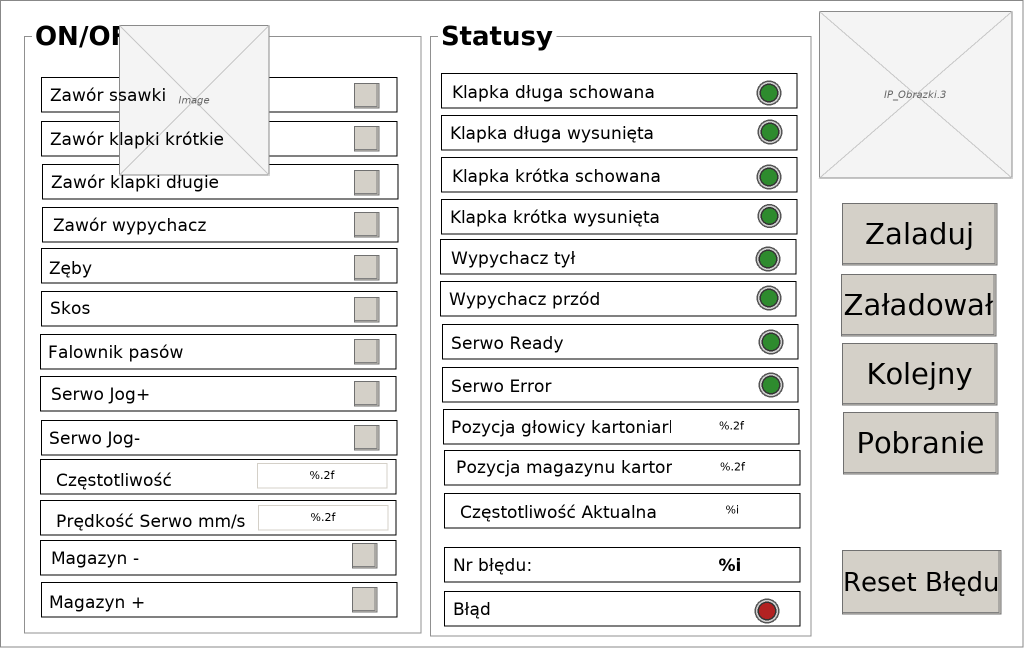
VISUALIZATION Kartoniarka  // 1024x648
    Rectangle (41,121 356x35)
    Rectangle (42,164 356x35)
    Rectangle (42,207 356x35)
    Rectangle (40,334 356x35)
    Rectangle (41,77 356x35)
    Rectangle (41,420 356x35)
    Rectangle (40,376 356x35)
    Rectangle (443,409 356x35)
    GroupBox (430,28 381x608), "Statusy"
        Rectangle (11,129 356x35)
        Rectangle (10,211 356x35)
        Label (18,384 330x30), "Pozycja głowicy kartoniarki"
        Rectangle (14,422 356x35)
        Label (23,424 330x30), "Pozycja magazynu kartonów"
    GroupBox (24,28 397x605), "ON/OFF"
        Rectangle (16,431 356x35)
        Rectangle (16,472 356x35)
        Textfield (234,477 130x25), "%.2f", text variable: gvl_hmi.J_VelK
            OnMouseClick: write the text variable via Edit
        Textfield (233,435 130x25), "%.2f", text variable: GVL_HMI.iFreqKartoniarkaMan
            OnMouseClick: write the text variable via Edit
        Button (330,397 25x25)
            tap GVL_HMI.bHmiJogKF
        Rectangle (17,554 356x35)
        Button (330,55 25x25), colour toggle: GVL_GLOBAL.zaw_ssawki_cewka
            tap GVL_HMI.przycisk_zaw_ssawki
        Button (330,311 25x25), colour toggle: GVL_GLOBAL.falownik_pasow_cewka
            tap GVL_HMI.przycisk_falownik_pasow
        Button (330,184 25x25), colour toggle: GVL_GLOBAL.zaw_wypychacz_cewka
            tap GVL_HMI.przycisk_zaw_wypychacz
        Button (330,142 25x25), colour toggle: GVL_GLOBAL.zaw_klap_dlug_cewka
            tap GVL_HMI.przycisk_zaw_klap_dlug
        Button (330,98 25x25), colour toggle: GVL_GLOBAL.zaw_klap_krot_cewka
            tap GVL_HMI.przycisk_zaw_klap_krot
        Rectangle (17,220 356x35)
        Rectangle (17,263 356x35)
        Label (23,265 209x30), "Skos"
        Button (330,269 25x25), colour toggle: GVL_GLOBAL.zaw_skos_cewka
            tap GVL_HMI.przycisk_zaw_skos
        Button (330,227 25x25), colour toggle: GVL_GLOBAL.zaw_zeby_cewka
            tap GVL_HMI.przycisk_zaw_zeby
        Button (330,353 25x25)
            tap GVL_HMI.bHmiJogKB
        Button (328,559 25x25)
            tap GVL_HMI.bHmiMagCcw
    Image (819,11 193x167), image: IP_Obrazki.3
    Button (842,343 155x62), "Kolejny"
        tap GVL_HMI.Nastepny_Karton
    Image (119,25 150x150)
    Rectangle (441,73 356x35)
    Label (447,76 230x30)
    Rectangle (441,115 356x35)
    Label (447,118 239x30), "Klapka długa wysunięta"
    Lamp1 (756,118 28x28), variable: GVL_IO.Kl_2_wyp, style: Lamp-Lamp1-Green
    Lamp1 (755,79 28x28), variable: GVL_IO.Kl_2_cof, style: Lamp-Lamp1-Green
    Label (449,77 239x30), "Klapka długa schowana"
    Rectangle (442,324 356x35)
    Rectangle (442,367 356x35)
    Label (48,167 209x30), "Zawór klapki długie"
    Label (47,119 239x30)
    Label (47,124 209x30), "Zawór klapki krótkie"
    Label (47,80 209x30), "Zawór ssawki"
    Label (50,210 209x30), "Zawór wypychacz"
    Label (45,337 209x30), "Falownik pasów"
    Label (53,465 209x30), "Częstotliwość"
    Label (448,328 239x30), "Serwo Ready"
    Lamp1 (757,328 28x28), variable: PRG_Kartoniarka.S_Power.Status, style: Lamp-Lamp1-Green
    Label (448,371 239x30), "Serwo Error"
    Lamp1 (757,371 28x28), variable: PRG_Kartoniarka.S_Power.Error, style: Lamp-Lamp1-Green
    Textfield (671,411 121x30), "%.2f", text variable: GVL_AXIS.stAxis1.NcToPlc.ActPos
    Label (48,379 209x30), "Serwo Jog+"
    Label (46,423 209x30), "Serwo Jog-"
    Label (447,160 230x30)
    Rectangle (441,199 356x35)
    Label (447,202 239x30), "Klapka krótka wysunięta"
    Lamp1 (756,202 27x28), variable: GVL_IO.Kl_1_wyp, style: Lamp-Lamp1-Green
    Lamp1 (755,163 28x28), variable: GVL_IO.Kl_1_cof, style: Lamp-Lamp1-Green
    Label (449,161 239x30), "Klapka krótka schowana"
    Label (446,242 230x30)
    Rectangle (440,281 356x35)
    Label (446,284 239x30), "Wypychacz przód"
    Lamp1 (755,284 28x28), variable: GVL_IO.Wyp_wys, style: Lamp-Lamp1-Green
    Lamp1 (754,245 28x28), variable: GVL_IO.Wyp_cof, style: Lamp-Lamp1-Green
    Label (448,243 239x30), "Wypychacz tył"
    Rectangle (444,493 356x35)
    Label (457,497 209x30), "Częstotliwość Aktualna"
    Textfield (672,495 121x30), "%i", text variable: GVL_HMI.iWydajnosc
    Textfield (672,452 121x30), "%.2f", text variable: GVL_AXIS.EC_Magazyn.NcToPlc.ActPos
    Label (53,506 209x30), "Prędkość Serwo mm/s"
    Rectangle (40,540 356x35)
    Button (352,543 25x25)
        tap GVL_HMI.bHmiMagCw
    Label (48,543 209x30), "Magazyn -"
    Label (46,587 209x30), "Magazyn +"
    Button (842,203 155x62), "Zaladuj"
        tap GVL_HMI.zaladuj
    Button (841,274 155x62), "Załadował"
        tap GVL_HMI.zaladowalem
    Button (843,412 155x62), "Pobranie"
        tap GVL_GLOBAL.Zabierz_Z_Kierownicy
    Label (46,253 209x30), "Zęby"
    Rectangle (444,547 356x35)
    Textfield (672,550 116x30), "%i", text variable: GVL_GLOBAL.Error_numb_kart
    Label (450,550 209x30), "Nr błędu:"
    Rectangle (444,591 356x35)
    Label (450,594 209x30), "Błąd"
    Button (842,550 159x64), "Reset Błędu"
        tap GVL_GLOBAL.Error_reset_kart
    Lamp1 (753,597 28x28), variable: GVL_GLOBAL.Error_ind_kart, style: Lamp-Lamp1-Red
END_VISUALIZATION

